(* IEC 61131-3 sources: SmartHomeNew/snapshots/2026-05-04, 69 files *)

(* ---- E_Behavior_Mode.dut ---- *)
TYPE E_Behavior_Mode :
(
    BEHAVIOR_HOME := 0,
    BEHAVIOR_AWAY := 1,
    BEHAVIOR_NIGHT := 2,
    BEHAVIOR_MAINTENANCE := 3
);
END_TYPE

(* ---- E_System_Reason_Code.dut ---- *)
{attribute 'strict'}
TYPE E_System_Reason_Code :
(
    REASON_NONE := 0,
    REASON_USER := 1,
    REASON_SAFETY := 2,
    REASON_AUTOMATION := 3,
    REASON_INTERNAL := 4,
    REASON_SCENARIO_VENT_BOOST := 5,
    REASON_USER_REQUEST := 6,
    REASON_SCENARIO_NIGHT := 7,
    REASON_DOMAIN_PROJECTION := 8
) USINT;
END_TYPE

(* ---- ST_Diagnostic_Event.dut ---- *)
{attribute 'pack_mode' := '1'}
TYPE ST_Diagnostic_Event :
STRUCT
    Code : UDINT;
    Severity : INT; // 1=info, 2=warning, 3=alarm, 4=critical
    Active : BOOL;
    Timestamp : UDINT;
    Source : INT; // producer/subsystem/index encoded by caller
END_STRUCT
END_TYPE

(* ---- ST_Operator_Zone_Rights.dut ---- *)
{attribute 'pack_mode' := '1'}
TYPE ST_Operator_Zone_Rights :
STRUCT
    operator_id : STRING(10);
    global_access_level : BYTE := 0;
    zone_masks : DWORD; // Битовая маска доступа к зонам (до 32 зон)
    last_modified : UDINT;
END_STRUCT
END_TYPE

(* ---- ST_System_Diagnostics.dut ---- *)
{attribute 'pack_mode' := '1'}
TYPE ST_System_Diagnostics :
STRUCT
    Freeze_Hardware_Event_Pending : BOOL;
    Freeze_Hardware_Event_Text : STRING(200);
    Backup_Pump_Fault : BOOL;
    Electric_Heater_Fault : BOOL;
    Backup_Pump_Recovered_After_Retry : BOOL;
    Electric_Heater_Recovered_After_Retry : BOOL;
    Backup_Pump_Out_Of_Service : BOOL;
    Electric_Heater_Out_Of_Service : BOOL;

    Pump_Exercise_Active : BOOL;
    Pump_Exercise_Failed : BOOL;
    Pump_Exercise_Last_Equipment : STRING(80);
    Pump_Exercise_Last_Result : STRING(120);
    Pump_Exercise_No_Feedback_Count : INT;
    Manifold_Pump_Exercise_Count : ARRAY[1..GVL_CONSTANTS.C_MAX_MANIFOLDS] OF UDINT;
    DHW_Heating_Pump_Exercise_Count : UDINT;
    DHW_Circ_Pump_Exercise_Count : UDINT;
    Backup_Pump_Exercise_Count : UDINT;
    Pump_Exercise_Event_Seq : UDINT;
    Pump_Exercise_Journal_1 : STRING(200);
    Pump_Exercise_Journal_2 : STRING(200);
    Pump_Exercise_Journal_3 : STRING(200);
    Pump_Exercise_Journal_Last_Seq : UDINT;

    Pump_Maintenance_Required : BOOL;
    Pump_Maintenance_Warning : BOOL;

    Manifold_Pump_Out_Of_Service : ARRAY[1..GVL_CONSTANTS.C_MAX_MANIFOLDS] OF BOOL;
    DHW_Heating_Pump_Out_Of_Service : BOOL;
    DHW_Circ_Pump_Out_Of_Service : BOOL;

    Maintenance_Last_Action : STRING(120);
    Operator_Action_Blocked : BOOL;
    Operator_Block_Reason : STRING(160);
    Operator_Last_Forbidden_Action : STRING(160);
    Operator_Journal_1 : STRING(200);
    Operator_Journal_2 : STRING(200);
    Operator_Journal_3 : STRING(200);
    Operator_Journal_Event_Seq : UDINT;
    Operator_Journal_Last_Seq : UDINT;

    Dangerous_Action_Pending_Confirm : BOOL;
    Dangerous_Action_Confirm_Text : STRING(160);
    Dangerous_Action_Confirm_Deadline_MS : UDINT;
    User_Access_Level_Active : INT;
    User_Access_Denied : BOOL;
    User_Access_Deny_Reason : STRING(160);

    Valve_Test_Mode_Active : BOOL;
    Valve_Test_Deadline_MS : UDINT;
    Valve_Test_Remaining_MS : UDINT;
    Valve_Test_Validation_OK : BOOL;
    Valve_Test_Validation_Text : STRING(160);
    Valve_Test_Forced_Close : BOOL;

    Water_Valve_Test_Mode_Active : BOOL;
    Water_Valve_Test_Deadline_MS : UDINT;
    Water_Valve_Test_Remaining_MS : UDINT;
    Water_Valve_Test_Validation_OK : BOOL;
    Water_Valve_Test_Validation_Text : STRING(160);
    Water_Valve_Test_Forced_Close : BOOL;
    Gas_Valve_Test_Mode_Active : BOOL;
    Gas_Valve_Test_Deadline_MS : UDINT;
    Gas_Valve_Test_Remaining_MS : UDINT;
    Gas_Valve_Test_Validation_OK : BOOL;
    Gas_Valve_Test_Validation_Text : STRING(160);
    Gas_Valve_Test_Forced_Close : BOOL;

    Active_Leak_Sensor_Index : INT;
    Active_Gas_Sensor_Index : INT;
    Active_Leak_Zone_Name : STRING(80);
    Active_Gas_Zone_Name : STRING(80);
    Water_Valve_Test_Context : STRING(160);
    Gas_Valve_Test_Context : STRING(160);

    Water_Recovery_Target_Zone_Index : INT;
    Gas_Recovery_Target_Zone_Index : INT;
    Water_Recovery_Selective_Allowed : BOOL;
    Gas_Recovery_Selective_Allowed : BOOL;
    Water_Recovery_Selective_Text : STRING(160);
    Gas_Recovery_Selective_Text : STRING(160);
    Water_Recovery_Physical_Active : BOOL;
    Water_Recovery_Physical_Zone_Name : STRING(80);

    Water_Zone_Open_Fault : ARRAY[1..32] OF BOOL;
    Water_Zone_Close_Fault : ARRAY[1..32] OF BOOL;
    Water_Valve_Exercise_Last_Zone : INT;
    Water_Valve_Exercise_Last_Result : STRING(160);
    Water_Zone_Critical_Close_Fault : ARRAY[1..32] OF BOOL;
    Water_Close_Fault_Active : BOOL;
    Water_Close_Fault_Zone_Name : STRING(80);
    Water_Close_Fault_Text : STRING(200);
    Water_Zone_Close_Retry_Active : ARRAY[1..32] OF BOOL;
    Water_Zone_Close_Retry_Count : ARRAY[1..32] OF INT;
    Water_Zone_Close_Recovered_After_Retry : ARRAY[1..32] OF BOOL;
    Water_Localization_Failed : BOOL;
    Water_Main_Shutdown_Recommended : BOOL;
    Water_Escalation_Text : STRING(200);
    Alarm_Event_Pulse : BOOL;
    Alarm_Event_Code : UDINT;
    Alarm_Event_Value : REAL;
    Sensor_Fault : BOOL;
    IO_Offline : BOOL;
    Subsystem_Degraded : BOOL;

    Manifold_Pressure_Fault : ARRAY[1..GVL_CONSTANTS.C_MAX_MANIFOLDS] OF BOOL;
    Manifold_Pressure_Diag_Code : ARRAY[1..GVL_CONSTANTS.C_MAX_MANIFOLDS] OF WORD;
    Manifold_Pressure_Fault_Active : BOOL;
    Manifold_Pressure_First_Fault_Index : INT;
    Manifold_Pressure_Fault_Text : STRING(160);

    Manifold_Current_Fault : ARRAY[1..GVL_CONSTANTS.C_MAX_MANIFOLDS] OF BOOL;
    Manifold_Current_Diag_Code : ARRAY[1..GVL_CONSTANTS.C_MAX_MANIFOLDS] OF WORD;
    Manifold_Current_Fault_Active : BOOL;
    Manifold_Current_First_Fault_Index : INT;
    Manifold_Current_Fault_Text : STRING(160);

    Manifold_Return_Temp_Fault : ARRAY[1..GVL_CONSTANTS.C_MAX_MANIFOLDS] OF BOOL;
    Manifold_Return_Temp_Diag_Code : ARRAY[1..GVL_CONSTANTS.C_MAX_MANIFOLDS] OF WORD;
    Manifold_Return_Temp_Fault_Active : BOOL;
    Manifold_Return_Temp_First_Fault_Index : INT;
    Manifold_Return_Temp_Fault_Text : STRING(160);

    Manifold_Sensor_Fault_Count : ARRAY[1..GVL_CONSTANTS.C_MAX_MANIFOLDS] OF INT;
    Manifold_Sensor_Out_Of_Service : ARRAY[1..GVL_CONSTANTS.C_MAX_MANIFOLDS] OF BOOL;
    Manifold_Sensor_Out_Of_Service_Active : BOOL;
    Manifold_Sensor_First_OOS_Index : INT;
    Manifold_Sensor_OOS_Text : STRING(160);
END_STRUCT
END_TYPE

(* ---- ST_Ventilation_Global_Config.dut ---- *)
{attribute 'pack_mode' := '1'}
TYPE ST_Ventilation_Global_Config :
STRUCT
    enable_ventilation : BOOL := TRUE;
    total_units : BYTE := 8;
    default_supply_speed : BYTE := 40;
    default_exhaust_speed : BYTE := 40;
    Degraded_Exhaust_Limit : BYTE := 30; // Ограничение вытяжки в режиме DEGRADED
    Scenario_Modes : ARRAY[1..GVL_CONSTANTS.C_MAX_SCENARIOS] OF ST_Ventilation_Scenario_Mode;
    wet_zone_to_exhaust_map : ARRAY[1..GVL_CONSTANTS.C_MAX_WET_ZONES] OF INT := [2, 3, 4, 5]; // Привязка мокрых зон к вытяжным вентиляторам
    pv3_exhaust_index : INT := 3; // Индекс вытяжного вентилятора ПВ-3
END_STRUCT
END_TYPE\n// VENT_POLICY_APPLIED
PolicyApplied : BOOL := TRUE;

(* ---- GVL_BEHAVIOR_ADAPT.gvl ---- *)
VAR_GLOBAL
    G_Behavior_Weights : ST_Behavior_Weights := (
        W_Comfort := 1.0,
        W_Night := 1.0,
        W_Preheat := 1.0,
        W_VentBoost := 1.0,
        W_AccessSecure := 1.0
    );

    G_Scenario_Stats : ARRAY[0..10] OF ST_Scenario_Stats;
    G_VentBoost_Zone_Adapt : ARRAY[1..GVL_CONSTANTS.C_MAX_ZONES] OF ST_Zone_Adapt_State;

    G_Adapt_Profile : E_Adapt_Profile := ADAPT_PROFILE_BALANCED;

    G_Adapt_Enabled : BOOL := TRUE;
    G_Adapt_Learning_Rate : REAL := 0.05;
    G_Adapt_Update_Threshold : INT := 5;

    G_Adapt_Min_Confidence : REAL := 0.30;
    G_Adapt_Default_Zone_Weight : REAL := 1.0;

    G_Confidence_Learning_Rate : REAL := 0.05;
    G_Decay_Factor : REAL := 0.995;

    G_Prev_Humidity : ARRAY[1..GVL_CONSTANTS.C_MAX_ZONES] OF REAL;
    G_Prev_Valid : ARRAY[1..GVL_CONSTANTS.C_MAX_ZONES] OF BOOL;
END_VAR
// >>> BULK_SYNC_ANCHOR: GVL_BEHAVIOR_ADAPT <<<

(* ---- GVL_COMMAND.gvl ---- *)
{attribute 'qualified_only'}
VAR_GLOBAL
    G_Gas_Valve_Close : BOOL := FALSE;
    G_Boiler_Stop : BOOL := FALSE;
    G_Supply_100_Req : BOOL := FALSE;
    G_Supply_80_Req : BOOL := FALSE;
    G_Vent_PV3_Boost : BOOL := FALSE;
    G_Exhaust_100_Req : BOOL := FALSE;
    G_Vent_Stop : BOOL := FALSE;
    G_Close_Valve_35 : BOOL := FALSE;
    G_Close_Valve_36 : BOOL := FALSE;
    G_Gate_Open : BOOL;
    G_Wicket_Open : BOOL;
    G_Lock_1_Open : BOOL;
    G_Lock_1_Close : BOOL;
    G_Lock_2_Open : BOOL;
    G_Lock_2_Close : BOOL;
    G_Reset_Errors : BOOL := FALSE;
    G_Scenario_Request : E_SCENARIO_TYPE := E_SCENARIO_TYPE.SCENARIO_NONE;
    G_Scenario_Request_Operator : E_SCENARIO_TYPE := E_SCENARIO_TYPE.SCENARIO_NONE;

    G_Arm_Req : BOOL;
    G_Disarm_Req : BOOL;
    G_PIN_Code : STRING(4);
    G_RFID_Tag : STRING(20);
    G_2FA_Code_In : STRING(6);
    G_Send_2FA_Req : BOOL;
    G_2FA_Code_Out : STRING(6);
    G_Lighting_Override : ARRAY[1..GVL_CONSTANTS.C_MAX_LIGHT_ZONES] OF BYTE;
    G_Blinds_Override : ARRAY[1..GVL_CONSTANTS.C_MAX_BLINDS] OF BYTE;
    G_Socket_Override : ARRAY[1..GVL_CONSTANTS.C_MAX_SOCKETS] OF BOOL;
    CMD_Set_Manifold_Pump_In_Service : ARRAY[1..GVL_CONSTANTS.C_MAX_MANIFOLDS] OF BOOL;
    CMD_Set_DHW_Heating_Pump_In_Service : BOOL;
    CMD_Set_DHW_Circ_Pump_In_Service : BOOL;
    CMD_Dangerous_Action_Confirm : BOOL;
    CMD_Dangerous_Action_Request : BOOL;
    CMD_User_Access_Level : INT := 0;
    CMD_Valve_Test_Open : BOOL;
    CMD_Valve_Test_Close : BOOL;
    CMD_Valve_Test_Confirm : BOOL;
    CMD_Water_Valve_Test_Open : BOOL;
    CMD_Water_Valve_Test_Close : BOOL;
    CMD_Water_Valve_Test_Confirm : BOOL;
    CMD_Gas_Valve_Test_Open : BOOL;
    CMD_Gas_Valve_Test_Close : BOOL;
    CMD_Gas_Valve_Test_Confirm : BOOL;
    CMD_Water_Selective_Recover : BOOL;
    CMD_Gas_Selective_Recover : BOOL;
END_VAR

(* ---- GVL_CONFIG.gvl ---- *)
{attribute 'qualified_only'}
VAR_GLOBAL
    // Subsystem Configurations
    G_Heating_Config : ST_Heating_Config; // Настройки системы отопления
    G_Ventilation_Config : ST_Ventilation_Config; // Настройки системы вентиляции
    G_DHW_Config : ST_DHW_Config; // Настройки горячего водоснабжения
    G_Security_Config : ST_Security_Global_Config; // Настройки системы безопасности
    G_Flood_Config : ST_Flood_Config; // Настройки системы защиты от протечек

    // HMI Configurations
    G_HMI_FloorHeating_Configs : ARRAY[1..GVL_CONSTANTS.C_MAX_HEATING_CIRCUITS] OF ST_FloorHeating_Circuit_Config; // Конфигурации контуров теплого пола
    G_Heating_Circuit_To_Zone : ARRAY[1..GVL_CONSTANTS.C_MAX_HEATING_CIRCUITS] OF INT := [1, 2, 3, 4, 5, 6, 7, 8, 9, 10, 11, 12, 13, 14, 15, 16]; // ВРЕМЕННО: circuit -> zone mapping, требует уточнения по фактической таблице помещений
    G_Wet_Zone_Map : ARRAY[1..32] OF BOOL; // Карта мокрых зон (TRUE = мокрая зона)
    G_HMI_Tariff_Settings : ST_Tariff_Config; // Настройки тарифов
    G_HMI_Vent_Global_Config : ST_Ventilation_Global_Config; // Глобальные настройки вентиляции
    G_HMI_Vent_Unit_Configs : ARRAY[1..GVL_CONSTANTS.C_MAX_VENT_UNITS] OF ST_Ventilation_Unit_Config; // Конфигурации отдельных вентустановок
    G_HMI_Scenario_Configs : ARRAY[1..GVL_CONSTANTS.C_MAX_SCENARIOS] OF ST_Scenario_Config; // Конфигурации сценариев
    G_HMI_Outdoor_Configs : ARRAY[1..GVL_CONSTANTS.C_MAX_OUTDOOR_ZONES] OF ST_Outdoor_Zone_Config; // Конфигурации зон уличного освещения
    G_HMI_Flood_Config : ST_Flood_Global_Config; // Глобальные настройки защиты от протечек
    G_HMI_Gas_Config : ST_Gas_Valve_Configuration; // Конфигурация системы газового контроля
    G_HMI_Sensor_Calibrations : ARRAY[1..GVL_CONSTANTS.C_MAX_CALIBRATIONS] OF ST_Sensor_Calibration_Record; // Данные калибровки датчиков
    G_HMI_User_Rules : ARRAY[1..GVL_CONSTANTS.C_MAX_RULES] OF ST_User_Rule; // Пользовательские правила (Rule Engine)

    // Sensor calibration pipeline
    G_Enable_Sensor_Calibration : BOOL := TRUE;
    G_Calib_Outdoor_Temp : ST_Sensor_Calibration_Record;
    G_Calib_Supply_Temps : ARRAY[1..GVL_CONSTANTS.C_MAX_SUPPLY_TEMPS] OF ST_Sensor_Calibration_Record;
    G_Calib_Room_Temps : ARRAY[1..GVL_CONSTANTS.C_MAX_ZONES] OF ST_Sensor_Calibration_Record;
    G_Calib_Floor_Temps : ARRAY[1..GVL_CONSTANTS.C_MAX_ZONES] OF ST_Sensor_Calibration_Record;
    G_Calib_CO2 : ARRAY[1..GVL_CONSTANTS.C_MAX_ZONES] OF ST_Sensor_Calibration_Record;
    G_Calib_Humidity : ARRAY[1..GVL_CONSTANTS.C_MAX_ZONES] OF ST_Sensor_Calibration_Record;
    G_Calib_Manifold_T_Supply : ARRAY[1..GVL_CONSTANTS.C_MAX_MANIFOLDS] OF ST_Sensor_Calibration_Record;
    G_Calib_Manifold_T_Return : ARRAY[1..GVL_CONSTANTS.C_MAX_MANIFOLDS] OF ST_Sensor_Calibration_Record;
    G_Calib_Methane : ARRAY[1..GVL_CONSTANTS.C_MAX_METHANE_SENSORS] OF ST_Sensor_Calibration_Record;
    G_Calib_CO : ARRAY[1..GVL_CONSTANTS.C_MAX_CO_SENSORS] OF ST_Sensor_Calibration_Record;

    // Конфигурация тестирования клапанов
    G_Valve_Test_Config : ARRAY[1..GVL_CONSTANTS.C_MAX_MANIFOLDS] OF ST_Valve_Test_Config;

    // HMI Commands & States
    G_HMI_Cleaning_Mode_Active : ARRAY[1..GVL_CONSTANTS.C_MAX_CLEANING_MODES] OF BOOL; // Режим уборки активен
    G_HMI_Cleaning_Mode_TimeLeft : ARRAY[1..GVL_CONSTANTS.C_MAX_CLEANING_MODES] OF UINT; // Оставшееся время режима уборки
    G_HMI_Admin_2FA_Enabled : BOOL := FALSE; // Включена ли 2FA для ADMIN
    G_HMI_Current_Operator_Factor2_Done : BOOL; // Второй фактор пройден
    G_HMI_Current_Operator_ID : STRING(10); // ID текущего оператора
    G_HMI_Manual_Gas_Valve_Open : BOOL; // Ручное открытие газового клапана
    G_HMI_Manual_Gas_Valve_Time : UDINT := 5; // Время ручного открытия
    G_HMI_Manual_Gas_Valve_TimeLeft : UDINT; // Оставшееся время ручного открытия
    G_HMI_Apply_Settings : BOOL; // Команда: Применить настройки
    G_HMI_Mute_Alarm : BOOL; // Команда: Временное отключение сирены
    G_HMI_Ack_Alarms : BOOL; // Команда: Квитировать все тревоги

    // Access Control Commands
    G_HMI_Gate_Open_Req : BOOL; // Запрос на открытие въездных ворот
    G_HMI_Wicket_Open_Req : BOOL; // Запрос на открытие калитки
    G_HMI_Lock_1_Open_Req : BOOL; // Разблокировка основного замка
    G_HMI_Lock_1_Close_Req : BOOL; // Блокировка основного замка
    G_HMI_Lock_2_Open_Req : BOOL; // Разблокировка доп. замка
    G_HMI_Lock_2_Close_Req : BOOL; // Блокировка доп. замка

    // HMI Settings
    G_HMI_Language : BYTE := 0; // 0=RU, 1=EN
    G_HMI_Brightness : BYTE := 80;
    G_HMI_Screen_Saver_Timeout : UDINT := 300; // сек

    // Сетевая безопасность
    G_Allowed_IPs : ARRAY[1..GVL_CONSTANTS.C_MAX_ALLOWED_IPS] OF STRING(15) := ['192.168.1.100','192.168.1.101','127.0.0.1','','']; // Разрешенные IP-адреса для шлюза

    G_Backup_Circulation_Pump_In_Service : BOOL := TRUE; // Резервный насос доступен для логики
    G_Electric_Heater_In_Service : BOOL := TRUE; // Электронагреватель доступен для логики
    G_Freeze_Hardware_Retry_Count : INT := 2; // Количество повторных попыток для anti-freeze hardware
    G_Freeze_Hardware_Retry_Delay_MS : UDINT := 5000; // Задержка между попытками повторного пуска
    G_Pump_Exercise_Enabled : BOOL := TRUE; // Разрешение периодической прокрутки насосов после простоя
    G_Pump_Exercise_Interval_MS : UDINT := 604800000; // 7 суток
    G_Pump_Exercise_Duration_MS : UDINT := 30000; // 30 сек
    G_Manifold_Pump_In_Service : ARRAY[1..GVL_CONSTANTS.C_MAX_MANIFOLDS] OF BOOL := [TRUE, TRUE, TRUE, TRUE, TRUE];
    G_Manifold_Priority : ARRAY[1..GVL_CONSTANTS.C_MAX_MANIFOLDS] OF INT := [3, 3, 2, 2, 1]; // 3=high, 2=normal, 1=low
    G_Manifold_Thermal_Weight : ARRAY[1..GVL_CONSTANTS.C_MAX_MANIFOLDS] OF REAL := [1.0, 1.0, 0.8, 0.8, 0.5];
    G_Max_Active_Manifolds : INT := 3; // energy-management limit for simultaneous active manifolds
    G_Max_Thermal_Budget : REAL := 6.0; // simplified manifold thermal budget units
    G_Policy_Min_Hold_MS : UDINT := 300000; // 5 min heating policy anti-oscillation hold
    G_DHW_Heating_Pump_In_Service : BOOL := TRUE;
    G_DHW_Circ_Pump_In_Service : BOOL := TRUE;
    G_Water_Valve_Exercise_Enabled : BOOL := TRUE;
    G_Water_Valve_Exercise_Interval_MS : UDINT := 604800000;
    G_Water_Valve_Exercise_Duration_MS : UDINT := 15000;
    G_Water_Valve_Exercise_Window_Start : TOD := TOD#04:00;
    G_Water_Valve_Exercise_Window_End : TOD := TOD#05:00;
    G_Water_Valve_Close_Retry_Count : INT := 2;
    G_Water_Valve_Close_Retry_Delay_MS : UDINT := 3000;
    // IO Mapping
    G_FloorTemp_Map : ARRAY[1..GVL_CONSTANTS.C_MAX_HEATING_CIRCUITS] OF INT := [1, 2, 3, 4, 5, 6, 7, 8, 9, 10, 11, 12, 13, 14, 15, 16];
    G_RoomTemp_Map : ARRAY[1..16] OF INT := [1, 2, 3, 4, 5, 6, 7, 8, 9, 10, 11, 12, 13, 14, 15, 16];
    G_Door_Map : ARRAY[1..GVL_CONSTANTS.C_MAX_DOOR_SENSORS] OF INT := [1, 2, 3, 4, 5, 6, 7, 8];
    G_Window_Map : ARRAY[1..16] OF INT := [9, 10, 11, 12, 13, 14, 15, 16, 17, 18, 19, 20, 21, 22, 23, 24];

    // Evacuation config
    C_MAX_LIGHT_ZONES : INT := 32; // fallback if not defined elsewhere
    G_Evac_Exit_Zones : ARRAY[1..32] OF BOOL; // зоны-выходы (TRUE = выход)
    G_Evac_Smoke_Zone_Map : ARRAY[1..GVL_CONSTANTS.C_MAX_SMOKE_SENSORS] OF INT; // Привязка дымовых датчиков к зонам эвакуации
    G_Evac_Leak_Zone_Map : ARRAY[1..GVL_CONSTANTS.C_MAX_FLOOD_SENSORS] OF INT; // Привязка датчиков протечки к зонам эвакуации
    G_Evac_Gas_Zone_Map : ARRAY[1..GVL_CONSTANTS.C_MAX_METHANE_SENSORS] OF INT; // Привязка газовых датчиков к зонам эвакуации
    G_Evac_Zone_Names : ARRAY[1..32] OF STRING(80); // Человекочитаемые имена зон (помещения/крыло/этаж/сторона)

END_VAR

VAR_GLOBAL CONSTANT
    C_MS_PER_SEC    : UDINT := GVL_CONSTANTS.C_MS_IN_SECOND; // Миллисекунд в секунду
    C_SEC_PER_MIN   : UDINT := 60; // Секунд в минуту
    C_MIN_PER_HOUR  : UDINT := 60; // Минут в часе
    C_MS_PER_MIN    : UDINT := GVL_CONSTANTS.C_MS_IN_MINUTE; // Миллисекунд в минуту
    C_MAX_RULES     : INT := 20; // Максимальное количество пользовательских правил
    C_ZONE_COUNT    : BYTE := 18; // Общее количество зон в системе

    // Коды ошибок
    ERR_PRESSURE_OUT_OF_RANGE : UDINT := 16#E004;
    ERR_HIGH_DELTA_T : UDINT := 16#E005;
    ERR_BOILER_OFFLINE : UDINT := 16#E006;
    ERR_BOILER_GENERAL_FAULT : UDINT := 16#E007;
    ERR_BOILER_NO_FLAME : UDINT := 16#E008;
    ERR_PUMP_NO_CURRENT : UDINT := 16#E009;
    ERR_PUMP_UNDERCURRENT : UDINT := 16#E00A;
    ERR_PUMP_OVERCURRENT : UDINT := 16#E00B;
    ERR_DELTA_T_LOW : UDINT := 16#E00C;
    ERR_DELTA_T_HIGH : UDINT := 16#E00D;
    ERR_DHW_IO_OFFLINE : UDINT := 16#E00E;
    ERR_DHW_TEMP_SENSOR_FAULT : UDINT := 16#E00F;
    ERR_DHW_PRESSURE_OUT_OF_RANGE : UDINT := 16#E010;
    ERR_DHW_PRESSURE_SENSOR_FAULT : UDINT := 16#E011;
    ERR_BACKUP_PUMP_OUT_OF_SERVICE : UDINT := 16#E012;
    ERR_ELECTRIC_HEATER_OUT_OF_SERVICE : UDINT := 16#E013;
    ERR_MANIFOLD_PUMP_OUT_OF_SERVICE : UDINT := 16#E014;
    ERR_DHW_HEATING_PUMP_OUT_OF_SERVICE : UDINT := 16#E015;
    ERR_DHW_CIRC_PUMP_OUT_OF_SERVICE : UDINT := 16#E016;
    ERR_FREEZE_HARDWARE_FAILED : UDINT := 16#E017;
END_VAR

(* ---- GVL_CONFIG_SIMULATION.gvl ---- *)
{attribute 'qualified_only'}
VAR_GLOBAL
    G_Simulation_Request : BOOL := FALSE;
    G_Simulation_Confirm : BOOL := FALSE;
    G_Simulation_Result_OK : BOOL := TRUE;
    G_Simulation_Error_Text : STRING(200) := '';
    G_Simulation_Last_Run_MS : UDINT := 0;
END_VAR

(* ---- GVL_CONFIG_VALIDATION.gvl ---- *)
{attribute 'qualified_only'}
VAR_GLOBAL
    G_Config_Valid : BOOL := TRUE;
    G_Config_Auto_Corrected : BOOL := FALSE;
    G_Config_Reset_To_Default_Done : BOOL := FALSE;
    G_Config_Last_Error_Text : STRING(200) := '';
    G_Config_Last_Action_Text : STRING(200) := '';
    G_Config_Last_Update_MS : UDINT := 0;
END_VAR

(* ---- GVL_DIAGNOSTICS_EXT.gvl ---- *)
{attribute 'qualified_only'}
VAR_GLOBAL
    // Health scores (0..1)
    G_Health_Heating : REAL := 1.0;
    G_Health_Safety : REAL := 1.0;
    G_Health_IO : REAL := 1.0;

    // Error counters
    G_Error_Count_Heating : UDINT := 0;
    G_Error_Count_Safety : UDINT := 0;
    G_Error_Count_IO : UDINT := 0;

    // Last error timestamps
    G_Last_Error_Time_Heating : UDINT := 0;
    G_Last_Error_Time_Safety : UDINT := 0;
    G_Last_Error_Time_IO : UDINT := 0;

    // Timing
    G_Last_Update_Time : UDINT := 0;

    // States
    G_Heating_State : INT := 0; // 0=OK,1=DEGRADED,2=CRITICAL
    G_Safety_State : INT := 0;
    G_IO_State : INT := 0;
END_VAR

(* ---- GVL_EVENT.gvl ---- *)
VAR_GLOBAL
    G_Event_Log : ARRAY[0..63] OF ST_EVENT;
    G_Event_Head : UINT;
    G_Event_ID_Counter : UDINT;
END_VAR

(* ---- GVL_INTENT_SAFETY.gvl ---- *)
VAR_GLOBAL
    // --- meta / traceability ---
    I_Source_Valid : BOOL := FALSE;
    I_Last_Update_Cycle : UDINT := 0;
    I_Last_Update_MS : UDINT := 0;

    // --- safety facts for arbitration ---
    I_Fire_Alarm_Active : BOOL := FALSE;
    I_Gas_Alarm_Active : BOOL := FALSE;
    I_Leak_Alarm_Active : BOOL := FALSE;
    I_CO_Warning_Active : BOOL := FALSE;
    I_System_Safe_Stop_Required : BOOL := FALSE;
    I_Freeze_Protection_Required : BOOL := FALSE;
    I_Evacuation_Mode_Active : BOOL := FALSE;

    // --- gas / boiler / ventilation constraints ---
    I_Gas_Close_Required : BOOL := FALSE;
    I_Boiler_Stop_Required : BOOL := FALSE;
    I_Vent_Stop_Required : BOOL := FALSE;
    I_Vent_Force_PV3_Boost : BOOL := FALSE;
    I_Vent_Force_Supply_100 : BOOL := FALSE;
    I_Vent_Force_Supply_80 : BOOL := FALSE;
    I_Vent_Force_Exhaust_100 : BOOL := FALSE;

    // --- water constraints ---
    I_Water_Main_Close_Required : BOOL := FALSE;
    I_Water_Zone_Close_Required : ARRAY[1..32] OF BOOL;
    I_Water_Selective_Recovery_Allowed : BOOL := FALSE;
    I_Water_Recovery_Target_Zone : INT := 0;

    // --- lock / evacuation constraints ---
    I_Lock_1_Force_Open : BOOL := FALSE;
    I_Lock_1_Force_Close_Block : BOOL := FALSE;
    I_Lock_2_Force_Open : BOOL := FALSE;
    I_Lock_2_Force_Close_Block : BOOL := FALSE;
END_VAR

(* ---- GVL_PRESENCE.gvl ---- *)
{attribute 'qualified_only'}
VAR_GLOBAL
    G_Any_Motion : BOOL := FALSE;
    G_Occupied : BOOL := TRUE;
    G_Auto_Away_Request : BOOL := FALSE;
    G_Last_Motion_TS : UDINT := 0;

    G_Zone_Occupied : ARRAY[1..GVL_CONSTANTS.C_MAX_ZONES] OF BOOL;
    G_Zone_Last_Motion_TS : ARRAY[1..GVL_CONSTANTS.C_MAX_ZONES] OF UDINT;
END_VAR

(* ---- GVL_Retain.gvl ---- *)
{attribute 'qualified_only'}
VAR_GLOBAL RETAIN
    G_Initialized : BOOL := FALSE; // Флаг инициализации retain-переменных

    // Энергонезависимая память (NVRAM) для хранения настроек и логов
    G_NVRAM_Data : ARRAY[0..12799] OF BYTE; // 100 * 128 = 12800 байт

    // Буфер черного ящика (100 записей)
    G_BlackBox_Buffer : ARRAY[0..GVL_CONSTANTS.C_MAX_BLACKBOX_RECORDS-1] OF ST_BlackBox_Record;
    G_BlackBox_LastIndex : INT;
    G_BlackBox_Frozen : BOOL;
    G_Presence_History : ARRAY[0..GVL_CONSTANTS.C_MAX_PRESENCE_HISTORY-1] OF WORD; // 168 часов * 6 записей в час = 1008 записей (битовая маска 16 ламп)

    // История событий
    G_History_Buffer : ARRAY[1..GVL_CONSTANTS.C_MAX_HISTORY_RECORDS] OF ST_History_Record;
    G_History_Write_Idx : INT := 1;
    G_History_Total_Events : UDINT;

    // Статистика котлов
    G_Boiler_Accumulated_MS : ARRAY[1..GVL_CONSTANTS.C_MAX_BOILERS] OF UDINT;
    G_Boiler_Work_Seconds : ARRAY[1..GVL_CONSTANTS.C_MAX_BOILERS] OF UDINT;

    // Результаты тестирования клапанов
    G_Valve_Test_Results : ARRAY[1..GVL_CONSTANTS.C_MAX_MANIFOLDS] OF BOOL;

    // ПИН-коды доступа (храним хэши CRC32 для безопасности)
    // 16#9BE3E0A3 - это CRC32 от строки '1234'
    G_Access_Codes : ARRAY[1..GVL_CONSTANTS.C_MAX_ACCESS_CODES] OF DWORD := [16#9BE3E0A3, 16#4A89A12D, 16#F4DBDF21, 16#90F59C65, 16#0972D346, 0, 0, 0, 0, 0];

    // Зарегистрированные RFID/NFC метки (строковое представление UID)
    G_RFID_Tags : ARRAY[1..GVL_CONSTANTS.C_MAX_ACCESS_CODES] OF STRING(20) := ['A1B2C3D4', 'E5F67890', '', '', '', '', '', '', '', ''];
END_VAR

(* ---- IValveController.st ---- *)
INTERFACE IValveController
METHOD OpenValve : BOOL
VAR_INPUT
    VI_Operator_ID : STRING(10);
    VI_Force : BOOL;
END_VAR
END_METHOD

METHOD CloseValve : BOOL
VAR_INPUT
    VI_Operator_ID : STRING(10);
    VI_Force : BOOL;
END_VAR
END_METHOD

METHOD GetStatus : BYTE
END_METHOD
END_INTERFACE

(* ---- FB_Analog_Validator.st ---- *)
FUNCTION_BLOCK FB_Analog_Validator
VAR_INPUT
    VI_Value : REAL;
    VI_Min_Valid : REAL;
    VI_Max_Valid : REAL;
    VI_Fallback_Mode : INT := 0; // 0: Hold last good, 1: Default value
    VI_Default_Value : REAL := 0.0;
END_VAR
VAR_OUTPUT
    VO_Value : REAL;
    VO_Error : BOOL;
END_VAR
VAR
    L_Last_Good_Value : REAL;
    L_First_Valid : BOOL := FALSE;
END_VAR

IF VI_Value >= VI_Min_Valid AND VI_Value <= VI_Max_Valid THEN
    VO_Error := FALSE;
    VO_Value := VI_Value;
    L_Last_Good_Value := VI_Value;
    L_First_Valid := TRUE;
ELSE
    VO_Error := TRUE;
    IF VI_Fallback_Mode = 1 OR NOT L_First_Valid THEN
        VO_Value := VI_Default_Value;
    ELSE
        VO_Value := L_Last_Good_Value;
    END_IF;
END_IF;
// >>> BULK_SYNC_ANCHOR: FB_Analog_Validator <<<

(* ---- FB_Device_Predictive_Diag.st ---- *)
FUNCTION_BLOCK FB_Device_Predictive_Diag
VAR_INPUT
    VI_Current_Value : REAL;      // Текущий ток или время
    VI_Nominal_Value : REAL;      // Эталонное значение
    VI_Is_Running    : BOOL;
    VI_Reset_Stats   : BOOL;
    VI_System_Time_MS: UDINT;     // Системное время (мс)
END_VAR
VAR_IN_OUT
    VIO_Health_Data  : ST_Device_Health;
END_VAR
VAR
    L_Prev_Running   : BOOL;
    L_Start_Time     : UDINT;
    L_Last_Calc_Time : UDINT;
    L_Elapsed_MS     : UDINT;
    L_Accumulated_MS : UDINT; // Накопленное время работы (мс)
    L_Timer_Running  : FB_System_Timer;
END_VAR

// 0. Сброс статистики
IF VI_Reset_Stats THEN
    VIO_Health_Data.Starts_Count := 0;
    VIO_Health_Data.Sample_Count := 0;
    VIO_Health_Data.Current_Sum := 0.0;
    VIO_Health_Data.Avg_Start_Current := 0.0;
    VIO_Health_Data.Health_Score := 100;
    VIO_Health_Data.Maintenance_Required := FALSE;
    VIO_Health_Data.Warning_Message := '';
    VIO_Health_Data.Last_Start_Current := 0.0;
    VIO_Health_Data.Total_Runtime_Hours := 0;
    L_Accumulated_MS := 0;
END_IF;

// 1. Счётчик пусков и замер пускового тока
IF VI_Is_Running AND NOT L_Prev_Running THEN
    VIO_Health_Data.Starts_Count := VIO_Health_Data.Starts_Count + 1;
    VIO_Health_Data.Last_Start_Current := VI_Current_Value;
    L_Start_Time := VI_System_Time_MS;
    L_Last_Calc_Time := VI_System_Time_MS;

    // Обновление среднего пускового тока
    VIO_Health_Data.Sample_Count := VIO_Health_Data.Sample_Count + 1;
    VIO_Health_Data.Current_Sum := VIO_Health_Data.Current_Sum + VI_Current_Value;
    VIO_Health_Data.Avg_Start_Current := VIO_Health_Data.Current_Sum / UDINT_TO_REAL(VIO_Health_Data.Sample_Count);

    // 2. Анализ отклонения пускового тока (п. 12.1 ТЗ)
    IF VI_Current_Value > (VI_Nominal_Value * 1.5) THEN
        VIO_Health_Data.Health_Score := TO_BYTE(LIMIT(0, TO_INT(VIO_Health_Data.Health_Score) - 5, 100));
    ELSIF VI_Current_Value > (VI_Nominal_Value * 1.2) THEN
        VIO_Health_Data.Health_Score := TO_BYTE(LIMIT(0, TO_INT(VIO_Health_Data.Health_Score) - 1, 100));
    ELSIF VI_Current_Value < (VI_Nominal_Value * 0.5) THEN
        VIO_Health_Data.Health_Score := TO_BYTE(LIMIT(0, TO_INT(VIO_Health_Data.Health_Score) - 2, 100));
    END_IF;
END_IF;

// 3. Анализ рабочего тока и наработки
IF VI_Is_Running THEN
    L_Elapsed_MS := (VI_System_Time_MS - L_Last_Calc_Time);
    L_Accumulated_MS := L_Accumulated_MS + L_Elapsed_MS;
    L_Last_Calc_Time := VI_System_Time_MS;

    // Обновляем наработку каждый час (3600000 мс)
    IF L_Accumulated_MS >= 3600000 THEN
        VIO_Health_Data.Total_Runtime_Hours := VIO_Health_Data.Total_Runtime_Hours + 1;
        L_Accumulated_MS := L_Accumulated_MS - 3600000;

        // Естественный износ: -1% здоровья каждые 1000 часов
        IF (VIO_Health_Data.Total_Runtime_Hours MOD 1000) = 0 THEN
            VIO_Health_Data.Health_Score := TO_BYTE(LIMIT(0, TO_INT(VIO_Health_Data.Health_Score) - 1, 100));
        END_IF;

        // Анализ рабочего тока (после пускового режима)
        IF (VI_System_Time_MS - L_Start_Time) > 10000 THEN // 10 секунд после пуска
            IF VI_Current_Value > (VI_Nominal_Value * 1.1) THEN
                // Повышенный рабочий ток - ускоренный износ (-1% в час)
                VIO_Health_Data.Health_Score := TO_BYTE(LIMIT(0, TO_INT(VIO_Health_Data.Health_Score) - 1, 100));
            END_IF;
        END_IF;
    END_IF;
END_IF;

// 4. Генерация предупреждения
IF VIO_Health_Data.Health_Score < 20 THEN
    VIO_Health_Data.Maintenance_Required := TRUE;
    VIO_Health_Data.Warning_Message := 'Критический износ: проверьте механику';
ELSIF VIO_Health_Data.Health_Score < 60 THEN
    VIO_Health_Data.Maintenance_Required := FALSE;
    VIO_Health_Data.Warning_Message := 'Предупреждение: повышенное трение';
ELSE
    VIO_Health_Data.Maintenance_Required := FALSE;
    VIO_Health_Data.Warning_Message := 'В норме';
END_IF;

L_Prev_Running := VI_Is_Running;

(* ---- FB_Diagnostics_Event_Manager.st ---- *)
FUNCTION_BLOCK FB_Diagnostics_Event_Manager
VAR_INPUT
    VI_Code : UDINT;
    VI_Severity : INT;
    VI_Active : BOOL;
    VI_Timestamp : UDINT;
    VI_Source : INT;
END_VAR
VAR_IN_OUT
    VIO_Events : ARRAY[1..50] OF ST_Diagnostic_Event;
    VIO_Count : INT;
END_VAR
VAR
    L_Index : INT;
    L_i : INT;
    L_Found_Index : INT;
    L_Was_Active : BOOL;
    L_Debounce_Index : INT;
    L_Oldest_Index : INT;
    L_Oldest_Time : UDINT;
    L_Stable_State : BOOL;

    L_Debounce_Used : ARRAY[1..50] OF BOOL;
    L_Debounce_Code : ARRAY[1..50] OF UDINT;
    L_Debounce_Source : ARRAY[1..50] OF INT;
    L_Debounce_Last_Input_State : ARRAY[1..50] OF BOOL;
    L_Debounce_Stable_State : ARRAY[1..50] OF BOOL;
    L_Debounce_Last_Change_Time : ARRAY[1..50] OF UDINT;
END_VAR

L_Found_Index := 0;
L_Was_Active := FALSE;
FOR L_i := 1 TO 50 DO
    IF (VIO_Events[L_i].Code = VI_Code) AND (VIO_Events[L_i].Source = VI_Source) THEN
        L_Found_Index := L_i;
        L_Was_Active := VIO_Events[L_i].Active;
        EXIT;
    END_IF;
END_FOR;

L_Debounce_Index := 0;
L_Oldest_Time := 16#FFFFFFFF;
L_Oldest_Index := 1;

FOR L_i := 1 TO 50 DO
    IF L_Debounce_Used[L_i] THEN
        IF (L_Debounce_Code[L_i] = VI_Code) AND (L_Debounce_Source[L_i] = VI_Source) THEN
            L_Debounce_Index := L_i;
            EXIT;
        END_IF;
        IF L_Debounce_Last_Change_Time[L_i] < L_Oldest_Time THEN
            L_Oldest_Time := L_Debounce_Last_Change_Time[L_i];
            L_Oldest_Index := L_i;
        END_IF;
    ELSE
        L_Debounce_Index := L_i;
        EXIT;
    END_IF;
END_FOR;

IF L_Debounce_Index = 0 THEN
    L_Debounce_Index := L_Oldest_Index;
END_IF;

IF NOT L_Debounce_Used[L_Debounce_Index] OR
   (L_Debounce_Code[L_Debounce_Index] <> VI_Code) OR
   (L_Debounce_Source[L_Debounce_Index] <> VI_Source) THEN
    L_Debounce_Used[L_Debounce_Index] := TRUE;
    L_Debounce_Code[L_Debounce_Index] := VI_Code;
    L_Debounce_Source[L_Debounce_Index] := VI_Source;
    L_Debounce_Last_Input_State[L_Debounce_Index] := VI_Active;
    L_Debounce_Stable_State[L_Debounce_Index] := FALSE;
    L_Debounce_Last_Change_Time[L_Debounce_Index] := VI_Timestamp;
END_IF;

IF VI_Active <> L_Debounce_Last_Input_State[L_Debounce_Index] THEN
    L_Debounce_Last_Input_State[L_Debounce_Index] := VI_Active;
    L_Debounce_Last_Change_Time[L_Debounce_Index] := VI_Timestamp;
END_IF;

IF (VI_Timestamp - L_Debounce_Last_Change_Time[L_Debounce_Index]) > 2000 THEN
    L_Debounce_Stable_State[L_Debounce_Index] := L_Debounce_Last_Input_State[L_Debounce_Index];
END_IF;

L_Stable_State := L_Debounce_Stable_State[L_Debounce_Index];

IF L_Stable_State THEN
    IF NOT L_Was_Active THEN
        L_Index := (VIO_Count MOD 50) + 1;
        VIO_Events[L_Index].Code := VI_Code;
        VIO_Events[L_Index].Severity := VI_Severity;
        VIO_Events[L_Index].Active := TRUE;
        VIO_Events[L_Index].Timestamp := VI_Timestamp;
        VIO_Events[L_Index].Source := VI_Source;
        VIO_Count := VIO_Count + 1;
    ELSIF L_Found_Index > 0 THEN
        VIO_Events[L_Found_Index].Severity := VI_Severity;
    END_IF;
ELSE
    IF L_Found_Index > 0 THEN
        VIO_Events[L_Found_Index].Active := FALSE;
    END_IF;
END_IF;

// >>> BULK_SYNC_ANCHOR: FB_Diagnostics_Event_Manager <<<

(* ---- FB_Diagnostics_RootCause.st ---- *)
FUNCTION_BLOCK FB_Diagnostics_RootCause
VAR_INPUT
    VI_Emergency_Stop : BOOL;
    VI_Gas_Safety : BOOL;
    VI_IO_Failsafe : BOOL;

    VI_Boiler_OT_Online : ARRAY[1..GVL_CONSTANTS.C_MAX_BOILERS] OF BOOL;
    VI_Boiler_Error : ARRAY[1..GVL_CONSTANTS.C_MAX_BOILERS] OF BOOL;
    VI_Boiler_Flame : ARRAY[1..GVL_CONSTANTS.C_MAX_BOILERS] OF BOOL;

    VI_Manifold_Pumps : ARRAY[1..GVL_CONSTANTS.C_MAX_MANIFOLDS] OF BOOL;
    VI_Manifold_Valves : ARRAY[1..GVL_CONSTANTS.C_MAX_MANIFOLDS] OF REAL;

    VI_Sensor_Error : BOOL;

    VI_Supply_Temps : ARRAY[1..GVL_CONSTANTS.C_MAX_MANIFOLDS] OF REAL;
    VI_Target_Supply : REAL;

    VI_Demand_Map : ARRAY[1..GVL_CONSTANTS.C_MAX_MANIFOLDS] OF BOOL;
END_VAR

VAR_OUTPUT
    VO_RootCause : E_Heating_RootCause;
    VO_Confidence : REAL;
END_VAR

VAR
    L_i : INT;
    L_AnyBoilerOnline : BOOL;
    L_AnyBoilerError : BOOL;
    L_AnyFlame : BOOL;
    L_AnyDemand : BOOL;
    L_AnyPumpOn : BOOL;
    L_AnyValveOpen : BOOL;
    L_LowSupply : BOOL;
END_VAR

// --- Safety ---
IF VI_Emergency_Stop THEN
    VO_RootCause := E_Heating_RootCause.RC_EMERGENCY_STOP;
    VO_Confidence := 1.0;
    RETURN;
END_IF;

IF VI_Gas_Safety THEN
    VO_RootCause := E_Heating_RootCause.RC_GAS_SAFETY;
    VO_Confidence := 1.0;
    RETURN;
END_IF;

IF VI_IO_Failsafe THEN
    VO_RootCause := E_Heating_RootCause.RC_IO_OFFLINE;
    VO_Confidence := 1.0;
    RETURN;
END_IF;

// --- Aggregate flags ---
L_AnyBoilerOnline := FALSE;
L_AnyBoilerError := FALSE;
L_AnyFlame := FALSE;

FOR L_i := 1 TO GVL_CONSTANTS.C_MAX_BOILERS DO
    IF VI_Boiler_OT_Online[L_i] THEN L_AnyBoilerOnline := TRUE; END_IF;
    IF VI_Boiler_Error[L_i] THEN L_AnyBoilerError := TRUE; END_IF;
    IF VI_Boiler_Flame[L_i] THEN L_AnyFlame := TRUE; END_IF;
END_FOR;

L_AnyDemand := FALSE;
L_AnyPumpOn := FALSE;
L_AnyValveOpen := FALSE;
L_LowSupply := FALSE;

FOR L_i := 1 TO GVL_CONSTANTS.C_MAX_MANIFOLDS DO
    IF VI_Demand_Map[L_i] THEN L_AnyDemand := TRUE; END_IF;
    IF VI_Manifold_Pumps[L_i] THEN L_AnyPumpOn := TRUE; END_IF;
    IF VI_Manifold_Valves[L_i] > 5.0 THEN L_AnyValveOpen := TRUE; END_IF;
    IF VI_Supply_Temps[L_i] < (VI_Target_Supply - 2.0) THEN L_LowSupply := TRUE; END_IF;
END_FOR;

// --- Boiler ---
IF NOT L_AnyBoilerOnline THEN
    VO_RootCause := E_Heating_RootCause.RC_BOILER_OFFLINE;
    VO_Confidence := 0.9;
    RETURN;
END_IF;

IF L_AnyBoilerError THEN
    VO_RootCause := E_Heating_RootCause.RC_BOILER_ERROR;
    VO_Confidence := 0.9;
    RETURN;
END_IF;

IF NOT L_AnyFlame THEN
    VO_RootCause := E_Heating_RootCause.RC_NO_FLAME;
    VO_Confidence := 0.8;
    RETURN;
END_IF;

// --- Hydraulics ---
IF L_AnyDemand THEN
    IF NOT L_AnyPumpOn THEN
        VO_RootCause := E_Heating_RootCause.RC_PUMP_FAILURE;
        VO_Confidence := 0.8;
        RETURN;
    END_IF;

    IF NOT L_AnyValveOpen THEN
        VO_RootCause := E_Heating_RootCause.RC_VALVES_CLOSED;
        VO_Confidence := 0.8;
        RETURN;
    END_IF;
END_IF;

// --- Thermal ---
IF L_AnyDemand AND L_LowSupply THEN
    VO_RootCause := E_Heating_RootCause.RC_NO_HEAT_TRANSFER;
    VO_Confidence := 0.7;
    RETURN;
END_IF;

// --- Sensors ---
IF VI_Sensor_Error THEN
    VO_RootCause := E_Heating_RootCause.RC_SENSOR_ERROR;
    VO_Confidence := 0.7;
    RETURN;
END_IF;

VO_RootCause := E_Heating_RootCause.RC_NONE;
VO_Confidence := 0.0;

END_FUNCTION_BLOCK

(* ---- FB_FloorHeating_Freeze_Protection.st ---- *)
FUNCTION_BLOCK FB_FloorHeating_Freeze_Protection
VAR_INPUT
    VI_Outdoor_Temp : REAL;
    VI_Threshold : REAL := 7.0;
END_VAR
VAR_IN_OUT
    VI_Floor_Temps : ARRAY[1..GVL_CONSTANTS.C_MAX_HEATING_CIRCUITS] OF REAL;
END_VAR
VAR_OUTPUT
    VO_Freeze_Alert : BOOL;
    VO_Pump_Force_On : BOOL;
END_VAR
VAR
    L_i : INT;
END_VAR

VO_Freeze_Alert := FALSE;
VO_Pump_Force_On := FALSE;

FOR L_i := 1 TO GVL_CONSTANTS.C_MAX_HEATING_CIRCUITS DO
    IF VI_Floor_Temps[L_i] < VI_Threshold THEN
        VO_Freeze_Alert := TRUE;
        VO_Pump_Force_On := TRUE;
        RETURN;
    END_IF;
END_FOR;

IF VI_Outdoor_Temp < -5.0 THEN
    VO_Pump_Force_On := TRUE;
END_IF;
END_FUNCTION_BLOCK

(* ---- FB_Heating_Execution_Core.st ---- *)
FUNCTION_BLOCK FB_Heating_Execution_Core
VAR_INPUT
    VI_System_Time_MS : UDINT;
    VI_Current_TOD : TOD;
    VI_Current_Day_Of_Week : UINT;
    VI_IsActivePLC : BOOL;
    VI_Outdoor_Temp : REAL;
    VI_Floor_Temps : ARRAY[1..GVL_CONSTANTS.C_MAX_HEATING_CIRCUITS] OF REAL;
    VI_Room_Temps : ARRAY[1..GVL_CONSTANTS.C_MAX_ZONES] OF REAL;
    VI_Config : ST_Heating_Config;
    VI_Zone_Configs : ARRAY[1..GVL_CONSTANTS.C_MAX_HEATING_CIRCUITS] OF ST_FloorHeating_Circuit_Config;
    VI_Tariff : ST_Tariff_Config;
    VI_Time_Of_Day_MS : UDINT;
    VI_Manifold_Pressures : ARRAY[1..GVL_CONSTANTS.C_MAX_MANIFOLDS] OF REAL;
    VI_Manifold_Currents : ARRAY[1..GVL_CONSTANTS.C_MAX_MANIFOLDS] OF REAL;
    VI_Manifold_Temps_Supply : ARRAY[1..GVL_CONSTANTS.C_MAX_MANIFOLDS] OF REAL;
    VI_Manifold_Temps_Return : ARRAY[1..GVL_CONSTANTS.C_MAX_MANIFOLDS] OF REAL;
    VI_Boiler_Flame_Status : ARRAY[1..GVL_CONSTANTS.C_MAX_BOILERS] OF BOOL;
    VI_Boiler_Error_Status : ARRAY[1..GVL_CONSTANTS.C_MAX_BOILERS] OF BOOL;
    VI_Boiler_OT_Online : ARRAY[1..GVL_CONSTANTS.C_MAX_BOILERS] OF BOOL;
    VI_Boiler_Modulation : ARRAY[1..GVL_CONSTANTS.C_MAX_BOILERS] OF REAL;
    VI_Rule_Actions : ARRAY[1..GVL_CONSTANTS.C_MAX_RULES] OF ST_Rule_Action;
    VI_IO_Modules_Online : ARRAY[1..GVL_CONSTANTS.C_MAX_MODULES] OF BOOL;
    VI_DHW_Heating_Demand : BOOL;
    VI_DHW_Target_Temp : REAL;
    VI_DHW_Temp : REAL;
    VI_DHW_Pressure : REAL;
    VI_DHW_Config : ST_DHW_Config;
    VI_Reset_Errors : BOOL;
    VI_System_Mode : E_System_Operating_Mode;
    VI_Emergency_Stop : BOOL;
    VI_Gas_Safety_Stop : BOOL;
    VI_Manifold_End_Switches : ARRAY[1..GVL_CONSTANTS.C_MAX_MANIFOLDS] OF BOOL;
    VI_Valve_Test_Config : ARRAY[1..GVL_CONSTANTS.C_MAX_MANIFOLDS] OF ST_Valve_Test_Config;
END_VAR
VAR_IN_OUT
    VIO_Manifold_Valves : ARRAY[1..GVL_CONSTANTS.C_MAX_MANIFOLDS] OF REAL;
    VIO_Manifold_Pumps : ARRAY[1..GVL_CONSTANTS.C_MAX_MANIFOLDS] OF BOOL;
    VIO_Zone_Valves : ARRAY[1..GVL_CONSTANTS.C_MAX_HEATING_CIRCUITS] OF BOOL;
    VIO_Boiler_OT_Enable : ARRAY[1..GVL_CONSTANTS.C_MAX_BOILERS] OF BOOL;
    VIO_Boiler_OT_Setpoint : ARRAY[1..GVL_CONSTANTS.C_MAX_BOILERS] OF REAL;
    VIO_Backup_Circulation_Pump : BOOL;
    VIO_Electric_Heater_Enable : BOOL;
    VIO_Freeze_Risk_Status : BOOL;
    VIO_Manifold_Status : ARRAY[1..GVL_CONSTANTS.C_MAX_MANIFOLDS] OF ST_Manifold_Status;
    VIO_Boiler_Status : ARRAY[1..GVL_CONSTANTS.C_MAX_BOILERS] OF ST_Boiler_Status;
    VIO_DHW_Heating_Pump : BOOL;
    VIO_DHW_Circ_Pump : BOOL;
    VIO_DHW_Status : ST_DHW_Status;
END_VAR
VAR
    fbHeatingManager : FB_Heating_System_Manager;
    fbDHWManager : FB_DHW_Manager;
END_VAR

// Pure execution core: calls heating and DHW managers.
// Does not apply command/allocation overrides.

fbHeatingManager(
    VI_System_Time_MS := VI_System_Time_MS,
    VI_IsActivePLC := VI_IsActivePLC,
    VI_Outdoor_Temp := VI_Outdoor_Temp,
    VI_Floor_Temps := VI_Floor_Temps,
    VI_Room_Temps := VI_Room_Temps,
    VI_Config := VI_Config,
    VI_Zone_Configs := VI_Zone_Configs,
    VI_Tariff := VI_Tariff,
    VI_Current_Hour := TO_UINT(VI_Time_Of_Day_MS / GVL_CONSTANTS.C_MS_IN_HOUR),
    VI_Manifold_Pressures := VI_Manifold_Pressures,
    VI_Manifold_Currents := VI_Manifold_Currents,
    VI_Manifold_Temps_Supply := VI_Manifold_Temps_Supply,
    VI_Manifold_Temps_Return := VI_Manifold_Temps_Return,
    VI_Boiler_Flame_Status := VI_Boiler_Flame_Status,
    VI_Boiler_Error_Status := VI_Boiler_Error_Status,
    VI_Boiler_OT_Online := VI_Boiler_OT_Online,
    VI_Boiler_Modulation := VI_Boiler_Modulation,
    VI_Rule_Actions := VI_Rule_Actions,
    VI_IO_Modules_Online := VI_IO_Modules_Online,
    VI_DHW_Heating_Demand := VI_DHW_Heating_Demand,
    VI_DHW_Target_Temp := VI_DHW_Target_Temp,
    VI_System_Mode := VI_System_Mode,
    VI_Emergency_Stop := VI_Emergency_Stop,
    VI_Gas_Safety_Stop := VI_Gas_Safety_Stop,
    VI_Manifold_End_Switches := VI_Manifold_End_Switches,
    VI_Valve_Test_Config := VI_Valve_Test_Config,
    VO_Manifold_Valves => VIO_Manifold_Valves,
    VO_Manifold_Pumps => VIO_Manifold_Pumps,
    VO_Zone_Valves => VIO_Zone_Valves,
    VO_Boiler_OT_Enable => VIO_Boiler_OT_Enable,
    VO_Boiler_OT_Setpoint => VIO_Boiler_OT_Setpoint,
    VO_Backup_Circulation_Pump => VIO_Backup_Circulation_Pump,
    VO_Electric_Heater_Enable => VIO_Electric_Heater_Enable,
    VO_Freeze_Risk_Status => VIO_Freeze_Risk_Status,
    VO_Status => VIO_Manifold_Status,
    VO_Boiler_Status => VIO_Boiler_Status
);

fbDHWManager(
    VI_System_Time_MS := VI_System_Time_MS,
    VI_Current_TOD := VI_Current_TOD,
    VI_IsActivePLC := VI_IsActivePLC,
    VI_Temp := VI_DHW_Temp,
    VI_Pressure := VI_DHW_Pressure,
    VI_Config := VI_DHW_Config,
    VI_Current_Day_Of_Week := VI_Current_Day_Of_Week,
    VI_IO_Modules_Online := VI_IO_Modules_Online,
    VI_Reset_Errors := VI_Reset_Errors,
    VI_Emergency_Stop := VI_Emergency_Stop,
    VI_System_Mode := VI_System_Mode,
    VO_Heating_Pump => VIO_DHW_Heating_Pump,
    VO_Circ_Pump => VIO_DHW_Circ_Pump,
    VO_Status => VIO_DHW_Status
);

END_FUNCTION_BLOCK
// >>> BULK_SYNC_ANCHOR: FB_Heating_Execution_Core <<<

(* ---- FB_Heating_Optimizer.st ---- *)
FUNCTION_BLOCK FB_Heating_Optimizer
VAR
    L_i : INT;
    L_Load : REAL;
    L_Total_Demand : REAL;
END_VAR

L_Total_Demand := 0.0;

// calculate total demand
FOR L_i := 1 TO GVL_CONSTANTS.C_MAX_ZONES DO
    L_Total_Demand := L_Total_Demand + ABS(GVL_HEATING_POLICY.G_Zone_Thermal_Demand[L_i]);
END_FOR;

GVL_HEATING_POLICY.G_Optimization_Load_Index := L_Total_Demand;

// normalize and optimize
FOR L_i := 1 TO GVL_CONSTANTS.C_MAX_ZONES DO

    IF L_Total_Demand > 0.01 THEN
        L_Load := ABS(GVL_HEATING_POLICY.G_Zone_Thermal_Demand[L_i]) / L_Total_Demand;
    ELSE
        L_Load := 0.0;
    END_IF;

    // priority score
    GVL_HEATING_POLICY.G_Zone_Optimization_Score[L_i] :=
        L_Load +
        (1.0 - GVL_HEATING_POLICY.G_Zone_Thermal_Model_Confidence[L_i]) * 0.2;

    // load balancing: reduce low priority zones
    IF GVL_HEATING_POLICY.G_Zone_Optimization_Score[L_i] < 0.2 THEN
        GVL_HEATING_POLICY.G_Zone_Thermal_Demand[L_i] :=
            GVL_HEATING_POLICY.G_Zone_Thermal_Demand[L_i] * 0.5;
    END_IF;

    // peak shaving
    IF L_Total_Demand > 5.0 THEN
        GVL_HEATING_POLICY.G_Zone_Thermal_Demand[L_i] :=
            GVL_HEATING_POLICY.G_Zone_Thermal_Demand[L_i] * 0.7;
        GVL_HEATING_POLICY.G_Optimization_Energy_Saving_Active := TRUE;
    END_IF;

END_FOR;

END_FUNCTION_BLOCK

(* ---- FB_Heating_Safe_State.st ---- *)
FUNCTION_BLOCK FB_Heating_Safe_State
VAR_INPUT
    VI_Block_Normal_Heating : BOOL;
    VI_IO_Failsafe_Active : BOOL;
    VI_Gas_Safety_Active : BOOL;
    VI_Freeze_Active : BOOL;
    VI_Freeze_Target_Supply : REAL;
    VI_Manifold_Temps_Supply : ARRAY[1..GVL_CONSTANTS.C_MAX_MANIFOLDS] OF REAL;
    VI_Boiler_Error_Status : ARRAY[1..GVL_CONSTANTS.C_MAX_BOILERS] OF BOOL;
    VI_Boiler_OT_Online : ARRAY[1..GVL_CONSTANTS.C_MAX_BOILERS] OF BOOL;
END_VAR
VAR_OUTPUT
    VO_Applied : BOOL;
    VO_Zone_Valves : ARRAY[1..GVL_CONSTANTS.C_MAX_HEATING_CIRCUITS] OF BOOL;
    VO_Manifold_Pumps : ARRAY[1..GVL_CONSTANTS.C_MAX_MANIFOLDS] OF BOOL;
    VO_Manifold_Valves : ARRAY[1..GVL_CONSTANTS.C_MAX_MANIFOLDS] OF REAL;
    VO_Boiler_OT_Enable : ARRAY[1..GVL_CONSTANTS.C_MAX_BOILERS] OF BOOL;
    VO_Boiler_OT_Setpoint : ARRAY[1..GVL_CONSTANTS.C_MAX_BOILERS] OF REAL;
    VO_Boiler_Status : ARRAY[1..GVL_CONSTANTS.C_MAX_BOILERS] OF ST_Boiler_Status;
    VO_Backup_Circulation_Pump : BOOL;
    VO_Electric_Heater_Enable : BOOL;
    VO_Freeze_Risk_Status : BOOL;
END_VAR
VAR
    L_i : INT;
    L_Min_Supply_Temp : REAL;
END_VAR

VO_Applied := VI_Block_Normal_Heating;
VO_Backup_Circulation_Pump := FALSE;
VO_Electric_Heater_Enable := FALSE;
VO_Freeze_Risk_Status := FALSE;

IF NOT VI_Block_Normal_Heating THEN
    RETURN;
END_IF;

FOR L_i := 1 TO GVL_CONSTANTS.C_MAX_HEATING_CIRCUITS DO
    VO_Zone_Valves[L_i] := FALSE;
END_FOR;

FOR L_i := 1 TO GVL_CONSTANTS.C_MAX_MANIFOLDS DO
    IF VI_IO_Failsafe_Active AND VI_Freeze_Active THEN
        VO_Manifold_Pumps[L_i] := TRUE;
        VO_Manifold_Valves[L_i] := 35.0;
    ELSE
        VO_Manifold_Pumps[L_i] := FALSE;
        VO_Manifold_Valves[L_i] := 0.0;
    END_IF;
END_FOR;

FOR L_i := 1 TO GVL_CONSTANTS.C_MAX_BOILERS DO
    VO_Boiler_OT_Enable[L_i] := FALSE;
    VO_Boiler_OT_Setpoint[L_i] := 0.0;
    VO_Boiler_Status[L_i].Warning := FALSE;
    VO_Boiler_Status[L_i].Error := TRUE;
END_FOR;

IF VI_Gas_Safety_Active AND VI_Freeze_Active THEN
    VO_Backup_Circulation_Pump := TRUE;
    L_Min_Supply_Temp := 1000.0;
    FOR L_i := 1 TO GVL_CONSTANTS.C_MAX_MANIFOLDS DO
        IF VI_Manifold_Temps_Supply[L_i] < L_Min_Supply_Temp THEN
            L_Min_Supply_Temp := VI_Manifold_Temps_Supply[L_i];
        END_IF;
    END_FOR;
    IF L_Min_Supply_Temp > 900.0 THEN
        L_Min_Supply_Temp := 0.0;
    END_IF;

    IF L_Min_Supply_Temp < (VI_Freeze_Target_Supply - 1.0) THEN
        VO_Electric_Heater_Enable := TRUE;
    ELSIF L_Min_Supply_Temp > (VI_Freeze_Target_Supply + 1.0) THEN
        VO_Electric_Heater_Enable := FALSE;
    END_IF;
    VO_Freeze_Risk_Status := TRUE;
END_IF;

IF VI_IO_Failsafe_Active AND VI_Freeze_Active THEN
    IF VI_Boiler_OT_Online[1] AND NOT VI_Boiler_Error_Status[1] THEN
        VO_Boiler_OT_Enable[1] := TRUE;
        VO_Boiler_OT_Setpoint[1] := VI_Freeze_Target_Supply;
    END_IF;
END_IF;

END_FUNCTION_BLOCK
// >>> BULK_SYNC_ANCHOR: FB_Heating_Safe_State <<<

(* ---- FB_Heating_Safety_Gate.st ---- *)
// ==============================================================================
// Heating safety gate helper
// ==============================================================================
FUNCTION_BLOCK FB_Heating_Safety_Gate
VAR_INPUT
    VI_System_Mode : E_System_Operating_Mode;
    VI_Emergency_Stop : BOOL;
    VI_Gas_Safety_Stop : BOOL;
    VI_IO_Failsafe_Active : BOOL;
    VI_Outdoor_Temp : REAL;
    VI_Freeze_Threshold : REAL;
END_VAR

VAR_IN_OUT
    VI_Floor_Temps : ARRAY[1..GVL_CONSTANTS.C_MAX_HEATING_CIRCUITS] OF REAL;
END_VAR

VAR_OUTPUT
    VO_Block_Normal_Heating : BOOL;
    VO_Gas_Safety_Active : BOOL;
    VO_Emergency_Safe_Stop_Active : BOOL;
    VO_IO_Failsafe_Active : BOOL;
    VO_Freeze_Mode_Active : BOOL;
    VO_Freeze_Target_Supply : REAL;
    VO_Outdoor_Temp_Valid : BOOL;
END_VAR

VAR
    L_i : INT;
    L_Outdoor_Temp_Safe : REAL;
END_VAR

VO_Gas_Safety_Active := VI_Gas_Safety_Stop;
VO_Emergency_Safe_Stop_Active := VI_Emergency_Stop OR (VI_System_Mode = E_System_Operating_Mode.MODE_SAFE_STOP);
VO_IO_Failsafe_Active := VI_IO_Failsafe_Active;

// REAL validity guard: NaN fails self-equality; extreme values are rejected as sensor faults.
VO_Outdoor_Temp_Valid := (VI_Outdoor_Temp = VI_Outdoor_Temp) AND (VI_Outdoor_Temp > -80.0) AND (VI_Outdoor_Temp < 80.0);
IF VO_Outdoor_Temp_Valid THEN
    L_Outdoor_Temp_Safe := VI_Outdoor_Temp;
ELSE
    L_Outdoor_Temp_Safe := 20.0;
    GVL_STATE.G_Heating_Sensor_Fault := TRUE;
END_IF;

VO_Block_Normal_Heating := VO_Gas_Safety_Active OR VO_Emergency_Safe_Stop_Active OR VO_IO_Failsafe_Active;
VO_Freeze_Mode_Active := (VI_System_Mode = E_System_Operating_Mode.MODE_FREEZE_PROTECTION) OR (L_Outdoor_Temp_Safe < -5.0);

FOR L_i := 1 TO GVL_CONSTANTS.C_MAX_HEATING_CIRCUITS DO
    IF VI_Floor_Temps[L_i] < 7.0 THEN
        VO_Freeze_Mode_Active := TRUE;
    END_IF;
END_FOR;

IF VO_Freeze_Mode_Active THEN
    VO_Freeze_Target_Supply := LIMIT(20.0, VI_Freeze_Threshold + 2.0, 35.0);
ELSE
    VO_Freeze_Target_Supply := 0.0;
END_IF;

// >>> BULK_SYNC_ANCHOR: FB_Heating_Safety_Gate <<<

(* ---- FB_HMI_Interface.st ---- *)
FUNCTION_BLOCK FB_HMI_Interface
VAR_INPUT
    VI_Severity   : E_System_Severity;
    VI_RootCause  : E_System_Root_Cause;
    VI_Status_Msg : STRING(200);
END_VAR

VAR_OUTPUT
    VO_HMI_Status_Text : STRING(200);
    VO_HMI_State_Code  : INT;
END_VAR

VO_HMI_Status_Text := VI_Status_Msg;

CASE VI_Severity OF
    E_System_Severity.SEV_NORMAL:
        VO_HMI_State_Code := 0;
    E_System_Severity.SEV_WARNING:
        VO_HMI_State_Code := 1;
    E_System_Severity.SEV_DEGRADED:
        VO_HMI_State_Code := 2;
    E_System_Severity.SEV_CRITICAL:
        VO_HMI_State_Code := 3;
END_CASE;
// >>> BULK_SYNC_ANCHOR: FB_HMI_Interface <<<

(* ---- FB_Lifetime_Manager.st ---- *)
FUNCTION_BLOCK FB_Lifetime_Manager
VAR_INPUT
    VI_System_Time_MS : UDINT;
    VI_Device_Active  : BOOL;
    VI_Device_ID      : BYTE;
    VI_Nominal_Hours : UDINT;
END_VAR

VAR_IN_OUT
    VIO_Status : ST_Lifetime_Status;
END_VAR

VAR
    L_Last_Time : UDINT;
    L_Prev_State : BOOL;
    L_Delta_MS : UDINT;
    L_Runtime_Accum_MS : UDINT;
    L_Remaining_Percent_UDINT : UDINT;
END_VAR

// === DELTA TIME ===
IF VI_System_Time_MS >= L_Last_Time THEN
    L_Delta_MS := VI_System_Time_MS - L_Last_Time;
ELSE
    // overflow
    L_Delta_MS := (4294967295 - L_Last_Time) + VI_System_Time_MS + 1;
END_IF;

L_Last_Time := VI_System_Time_MS;

// === START COUNT ===
IF VI_Device_Active AND NOT L_Prev_State THEN
    VIO_Status.start_count := VIO_Status.start_count + 1;
END_IF;

L_Prev_State := VI_Device_Active;

// === RUNTIME ACCUMULATION ===
IF VI_Device_Active THEN
    L_Runtime_Accum_MS := L_Runtime_Accum_MS + L_Delta_MS;

    WHILE L_Runtime_Accum_MS >= 3600000 DO
        VIO_Status.runtime_hours := VIO_Status.runtime_hours + 1;
        L_Runtime_Accum_MS := L_Runtime_Accum_MS - 3600000;
    END_WHILE;
END_IF;

// === BASIC LIFETIME ESTIMATION ===
IF VI_Nominal_Hours > 0 THEN
    IF VIO_Status.runtime_hours >= VI_Nominal_Hours THEN
        VIO_Status.remaining_hours := 0;
        VIO_Status.remaining_percent := 0;
    ELSE
        VIO_Status.remaining_hours := VI_Nominal_Hours - VIO_Status.runtime_hours;
        L_Remaining_Percent_UDINT := (VIO_Status.remaining_hours * 100) / VI_Nominal_Hours;

        IF L_Remaining_Percent_UDINT > 100 THEN
            L_Remaining_Percent_UDINT := 100;
        END_IF;

        VIO_Status.remaining_percent := UDINT_TO_BYTE(L_Remaining_Percent_UDINT);
    END_IF;
ELSE
    VIO_Status.remaining_hours := 0;
    VIO_Status.remaining_percent := 0;
END_IF;

VIO_Status.maintenance_required := VIO_Status.remaining_percent <= GVL_Lifetime.G_Maintenance_Threshold_Percent;

// === BASIC FLAGS ===
VIO_Status.device_id := VI_Device_ID;
VIO_Status.last_calc_timestamp := VI_System_Time_MS;

END_FUNCTION_BLOCK

(* ---- FB_Maintenance_Access.st ---- *)
FUNCTION_BLOCK FB_Maintenance_Access
VAR_INPUT
    VI_System_Time : UDINT;
    VI_Activate    : BOOL;
    VI_Duration    : UDINT := 60; // мин
END_VAR
VAR_OUTPUT
    VO_Active      : BOOL;
    VO_Time_Left   : UDINT;
END_VAR
VAR
    L_Start_Time   : UDINT;
    L_elapsed      : UDINT;
END_VAR

IF VI_Activate AND NOT VO_Active THEN
    VO_Active := TRUE;
    L_Start_Time := VI_System_Time;
END_IF;

IF VO_Active THEN
    L_elapsed := (SEL(VI_System_Time >= L_Start_Time, VI_System_Time - L_Start_Time, (4294967295 - L_Start_Time) + VI_System_Time + 1)) / GVL_CONSTANTS.C_MS_IN_MINUTE;
    IF L_elapsed >= VI_Duration THEN
        VO_Active := FALSE;
        VO_Time_Left := 0;
    ELSE
        VO_Time_Left := VI_Duration - L_elapsed;
    END_IF;
ELSE
    VO_Time_Left := 0;
END_IF;

(* ---- FB_Mode_Manager.st ---- *)
FUNCTION_BLOCK FB_Mode_Manager

VAR_INPUT
    VI_Is_Night : BOOL;
    VI_Away_Request : BOOL;
    VI_Maintenance_Request : BOOL;
    VI_System_Time_MS : UDINT;
END_VAR

VAR_OUTPUT
    VO_Mode : E_Behavior_Mode;
    VO_Mode_Code : UDINT;
END_VAR

// default
VO_Mode := BEHAVIOR_HOME;
VO_Mode_Code := 0;

// priority-based transitions
IF VI_Maintenance_Request THEN
    VO_Mode := BEHAVIOR_MAINTENANCE;
    VO_Mode_Code := 300;
ELSIF VI_Away_Request THEN
    VO_Mode := BEHAVIOR_AWAY;
    VO_Mode_Code := 200;
ELSIF VI_Is_Night THEN
    VO_Mode := BEHAVIOR_NIGHT;
    VO_Mode_Code := 100;
END_IF;

(* ---- FB_Persist_Pipeline.st ---- *)
FUNCTION_BLOCK FB_Persist_Pipeline
VAR_INPUT
    VI_PersistStruct : ST_Persist;
    VI_System_Time_MS : UDINT;
    VI_IsActivePLC : BOOL;
END_VAR
VAR_IN_OUT
    VIO_Apply_Settings : BOOL;
    VIO_Persist_Buffer : ARRAY[0..4] OF BYTE;
    VIO_Last_Written_Persist_Buffer : ARRAY[0..4] OF BYTE;
    VIO_Last_Persist_Write_MS : UDINT;
END_VAR
VAR_OUTPUT
    VO_NVRAM_Cmd : BYTE;
    VO_NVRAM_Offset : UDINT;
    VO_NVRAM_Done : BOOL;
    VO_NVRAM_Err : BOOL;
    VO_NVRAM_ErrID : UDINT;
END_VAR
VAR
    fbNVRAMManager : FB_NVRAM_Manager;
    L_Persist_Buffer_Changed : BOOL;
END_VAR

// === SERIALIZE PERSIST STRUCT → BUFFER ===

// System Mode
VIO_Persist_Buffer[0] := TO_BYTE(TO_INT(VI_PersistStruct.System_Mode));

// Gas
IF VI_PersistStruct.Safety_Gas_Latched THEN
    VIO_Persist_Buffer[1] := BYTE#1;
ELSE
    VIO_Persist_Buffer[1] := BYTE#0;
END_IF;

// Smoke
IF VI_PersistStruct.Safety_Smoke_Latched THEN
    VIO_Persist_Buffer[2] := BYTE#1;
ELSE
    VIO_Persist_Buffer[2] := BYTE#0;
END_IF;

// Leak
IF VI_PersistStruct.Safety_Leak_Latched THEN
    VIO_Persist_Buffer[3] := BYTE#1;
ELSE
    VIO_Persist_Buffer[3] := BYTE#0;
END_IF;

// DHW Pump
IF VI_PersistStruct.DHW_Heating_Pump THEN
    VIO_Persist_Buffer[4] := BYTE#1;
ELSE
    VIO_Persist_Buffer[4] := BYTE#0;
END_IF;

// === END SERIALIZE ===

L_Persist_Buffer_Changed :=
    (VIO_Persist_Buffer[0] <> VIO_Last_Written_Persist_Buffer[0]) OR
    (VIO_Persist_Buffer[1] <> VIO_Last_Written_Persist_Buffer[1]) OR
    (VIO_Persist_Buffer[2] <> VIO_Last_Written_Persist_Buffer[2]) OR
    (VIO_Persist_Buffer[3] <> VIO_Last_Written_Persist_Buffer[3]) OR
    (VIO_Persist_Buffer[4] <> VIO_Last_Written_Persist_Buffer[4]);

VO_NVRAM_Cmd := 0;
VO_NVRAM_Offset := 0;

IF VIO_Apply_Settings THEN
    // explicit config apply requests a controlled write
    // keep flag set until successful write confirmation
    VO_NVRAM_Cmd := 1;

ELSIF L_Persist_Buffer_Changed THEN
    // controlled write: no more often than once per 60 seconds
    IF (VIO_Last_Persist_Write_MS = 0) OR
       ((VI_System_Time_MS - VIO_Last_Persist_Write_MS) >= 60000) THEN
        VO_NVRAM_Cmd := 1;
    END_IF;
END_IF;

fbNVRAMManager(
    VI_Command := VO_NVRAM_Cmd,
    VI_Offset := VO_NVRAM_Offset,
    VI_DataRef := VIO_Persist_Buffer[0],
    VI_DataSize := 5,
    VI_System_Time_MS := VI_System_Time_MS,
    VI_Operator_ID := 'SYSTEM',
    VI_IsActivePLC := VI_IsActivePLC,
    VI_TwoPersonConfirmation := FALSE,
    VO_Done => VO_NVRAM_Done,
    VO_Error => VO_NVRAM_Err,
    VO_ErrorID => VO_NVRAM_ErrID
);

IF (VO_NVRAM_Cmd = 1) AND VO_NVRAM_Done AND NOT VO_NVRAM_Err THEN
    VIO_Last_Written_Persist_Buffer[0] := VIO_Persist_Buffer[0];
    VIO_Last_Written_Persist_Buffer[1] := VIO_Persist_Buffer[1];
    VIO_Last_Written_Persist_Buffer[2] := VIO_Persist_Buffer[2];
    VIO_Last_Written_Persist_Buffer[3] := VIO_Persist_Buffer[3];
    VIO_Last_Written_Persist_Buffer[4] := VIO_Persist_Buffer[4];
    VIO_Last_Persist_Write_MS := VI_System_Time_MS;
    VIO_Apply_Settings := FALSE;
END_IF;
END_FUNCTION_BLOCK

(* ---- FB_PID_Controller.st ---- *)
FUNCTION_BLOCK FB_PID_Controller
VAR_INPUT
    VI_SetPoint : REAL;
    VI_ProcessValue : REAL;
    VI_Kp : REAL;
    VI_Tn : REAL;
    VI_Tv : REAL;
    VI_Y_Min : REAL := REAL#0.0;
    VI_Y_Max : REAL := REAL#100.0;
    VI_Manual_Mode : BOOL;
    VI_Manual_Value : REAL;
    VI_Deadband : REAL := REAL#0.1;
    VI_Cycle_Time_S : REAL := REAL#0.01;
    VI_Reset : BOOL;
END_VAR
VAR_OUTPUT
    VO_Output : REAL;
    VO_Error : REAL;
    VO_Limiting : BOOL;
END_VAR
VAR
    L_Integral_Sum : REAL;
    L_Prev_Error : REAL;
    L_Derivative : REAL;
    L_P_Term : REAL;
    L_I_Candidate : REAL;
    L_D_Term : REAL;
    L_Output_Predicted : REAL;
    L_Output_Raw : REAL;
    L_Cycle_Time_Safe : REAL;
END_VAR

L_Cycle_Time_Safe := VI_Cycle_Time_S;
IF L_Cycle_Time_Safe <= REAL#0.0 THEN
    L_Cycle_Time_Safe := REAL#0.01;
END_IF;

VO_Error := VI_SetPoint - VI_ProcessValue;
IF ABS(VO_Error) < VI_Deadband THEN
    VO_Error := REAL#0.0;
END_IF;

IF VI_Reset THEN
    L_Integral_Sum := REAL#0.0;
    L_Prev_Error := REAL#0.0;
    VO_Output := LIMIT(VI_Y_Min, REAL#0.0, VI_Y_Max);
    VO_Limiting := FALSE;
    RETURN;
END_IF;

L_P_Term := VI_Kp * VO_Error;

IF VI_Tv > REAL#0.0 THEN
    L_Derivative := (VO_Error - L_Prev_Error) / L_Cycle_Time_Safe;
    L_D_Term := VI_Kp * VI_Tv * L_Derivative;
ELSE
    L_Derivative := REAL#0.0;
    L_D_Term := REAL#0.0;
END_IF;

IF VI_Manual_Mode THEN
    VO_Output := LIMIT(VI_Y_Min, VI_Manual_Value, VI_Y_Max);
    L_Integral_Sum := VO_Output - L_P_Term - L_D_Term;
    L_Prev_Error := VO_Error;
    VO_Limiting := (VO_Output <= VI_Y_Min) OR (VO_Output >= VI_Y_Max);
    RETURN;
END_IF;

IF VI_Tn > REAL#0.0 THEN
    L_I_Candidate := L_Integral_Sum + ((VI_Kp / VI_Tn) * VO_Error * L_Cycle_Time_Safe);
ELSE
    L_I_Candidate := L_Integral_Sum;
END_IF;

L_Output_Predicted := L_P_Term + L_I_Candidate + L_D_Term;

// Anti-windup: accept the new integral only if it does not push the output farther into saturation.
IF VI_Tn > REAL#0.0 THEN
    IF (L_Output_Predicted > VI_Y_Max) AND (VO_Error > REAL#0.0) THEN
        // hold integral
    ELSIF (L_Output_Predicted < VI_Y_Min) AND (VO_Error < REAL#0.0) THEN
        // hold integral
    ELSE
        L_Integral_Sum := L_I_Candidate;
    END_IF;
END_IF;

L_Output_Raw := L_P_Term + L_Integral_Sum + L_D_Term;
VO_Output := LIMIT(VI_Y_Min, L_Output_Raw, VI_Y_Max);
VO_Limiting := (L_Output_Raw > VI_Y_Max) OR (L_Output_Raw < VI_Y_Min);
L_Prev_Error := VO_Error;

// >>> BULK_SYNC_ANCHOR: FB_PID_Controller <<<
END_FUNCTION_BLOCK

(* ---- FB_Rule_Engine.st ---- *)
FUNCTION_BLOCK FB_Rule_Engine
VAR_INPUT
    VI_System_Time_MS : UDINT;
    VI_IsActivePLC : BOOL;
    VI_Security_Armed : BOOL;
    VI_Current_Time : TOD;
    VI_Day_Of_Week : INT;
END_VAR
VAR_IN_OUT
    VI_Rules : ARRAY[1..GVL_CONSTANTS.C_MAX_RULES] OF ST_User_Rule;
    VI_Indoor_Temps : ARRAY[1..16] OF REAL;
    VI_Floor_Temps : ARRAY[1..GVL_CONSTANTS.C_MAX_HEATING_CIRCUITS] OF REAL;
    VI_Humidities : ARRAY[1..16] OF REAL;
    VI_CO2_Levels : ARRAY[1..16] OF REAL;
    VI_Motion_Sensors : ARRAY[1..16] OF BOOL;
    VI_Door_Sensors : ARRAY[1..GVL_CONSTANTS.C_MAX_DOOR_SENSORS] OF BOOL;
    VI_Window_Sensors : ARRAY[1..16] OF BOOL;
    VI_Water_Sensors : ARRAY[1..GVL_CONSTANTS.C_MAX_FLOOD_SENSORS] OF BOOL;
    VI_Smoke_Sensors : ARRAY[1..GVL_CONSTANTS.C_MAX_SMOKE_SENSORS] OF BOOL;
    VI_Methane_Sensors : ARRAY[1..GVL_CONSTANTS.C_MAX_METHANE_SENSORS] OF REAL;
    VI_CO_Sensors : ARRAY[1..GVL_CONSTANTS.C_MAX_CO_SENSORS] OF REAL;
END_VAR
VAR_OUTPUT
    VO_Preheat_Request : BOOL;
    VO_Actions : ARRAY[1..GVL_CONSTANTS.C_MAX_RULES] OF ST_Rule_Action;
END_VAR
VAR
    L_i : INT;
    L_Condition_Met : BOOL;
    L_Current_Value : REAL;
    L_Triggers : ARRAY[1..GVL_CONSTANTS.C_MAX_RULES] OF R_TRIG;
    L_Trigger_Count : ARRAY[1..GVL_CONSTANTS.C_MAX_RULES] OF UINT;
    L_Last_Reset_Time : UDINT;
    L_Elapsed_Time : UDINT;
END_VAR

IF NOT VI_IsActivePLC THEN RETURN; END_IF;

VO_Preheat_Request := FALSE;

L_Elapsed_Time := SEL(VI_System_Time_MS >= L_Last_Reset_Time, VI_System_Time_MS - L_Last_Reset_Time, (4294967295 - L_Last_Reset_Time) + VI_System_Time_MS + 1);

IF L_Elapsed_Time >= GVL_CONSTANTS.C_MS_IN_MINUTE THEN
    L_Last_Reset_Time := VI_System_Time_MS;
    FOR L_i := 1 TO GVL_CONSTANTS.C_MAX_RULES DO
        L_Trigger_Count[L_i] := 0;
    END_FOR;
END_IF;

FOR L_i := 1 TO GVL_CONSTANTS.C_MAX_RULES DO

    VO_Actions[L_i].Active := FALSE;
    IF VI_Rules[L_i].Enabled THEN
        L_Condition_Met := FALSE;
        L_Current_Value := 0.0;

        IF VI_Rules[L_i].Condition_Target_ID > 0 THEN
            CASE VI_Rules[L_i].Condition_Type OF
                E_Rule_Condition_Type.COND_AIR_TEMP: IF VI_Rules[L_i].Condition_Target_ID <= 16 THEN L_Current_Value := VI_Indoor_Temps[VI_Rules[L_i].Condition_Target_ID]; END_IF;
                E_Rule_Condition_Type.COND_FLOOR_TEMP: IF VI_Rules[L_i].Condition_Target_ID <= GVL_CONSTANTS.C_MAX_HEATING_CIRCUITS THEN L_Current_Value := VI_Floor_Temps[VI_Rules[L_i].Condition_Target_ID]; END_IF;
                E_Rule_Condition_Type.COND_HUMIDITY: IF VI_Rules[L_i].Condition_Target_ID <= 16 THEN L_Current_Value := VI_Humidities[VI_Rules[L_i].Condition_Target_ID]; END_IF;
                E_Rule_Condition_Type.COND_CO2: IF VI_Rules[L_i].Condition_Target_ID <= 16 THEN L_Current_Value := VI_CO2_Levels[VI_Rules[L_i].Condition_Target_ID]; END_IF;
                E_Rule_Condition_Type.COND_MOTION: IF VI_Rules[L_i].Condition_Target_ID <= 16 THEN L_Current_Value := SEL(VI_Motion_Sensors[VI_Rules[L_i].Condition_Target_ID], 0.0, 1.0); END_IF;
                E_Rule_Condition_Type.COND_DOOR_WINDOW:
                    IF VI_Rules[L_i].Condition_Target_ID <= GVL_CONSTANTS.C_MAX_DOOR_SENSORS THEN
                        L_Current_Value := SEL(VI_Door_Sensors[VI_Rules[L_i].Condition_Target_ID] OR VI_Window_Sensors[VI_Rules[L_i].Condition_Target_ID], 0.0, 1.0);
                    ELSIF VI_Rules[L_i].Condition_Target_ID <= 16 THEN
                        L_Current_Value := SEL(VI_Window_Sensors[VI_Rules[L_i].Condition_Target_ID], 0.0, 1.0);
                    END_IF;
                E_Rule_Condition_Type.COND_FLOOD: IF VI_Rules[L_i].Condition_Target_ID <= GVL_CONSTANTS.C_MAX_FLOOD_SENSORS THEN L_Current_Value := SEL(VI_Water_Sensors[VI_Rules[L_i].Condition_Target_ID], 0.0, 1.0); END_IF;
                E_Rule_Condition_Type.COND_SMOKE: IF VI_Rules[L_i].Condition_Target_ID <= GVL_CONSTANTS.C_MAX_SMOKE_SENSORS THEN L_Current_Value := SEL(VI_Smoke_Sensors[VI_Rules[L_i].Condition_Target_ID], 0.0, 1.0); END_IF;
                E_Rule_Condition_Type.COND_METHANE: IF VI_Rules[L_i].Condition_Target_ID <= GVL_CONSTANTS.C_MAX_METHANE_SENSORS THEN L_Current_Value := VI_Methane_Sensors[VI_Rules[L_i].Condition_Target_ID]; END_IF;
                E_Rule_Condition_Type.COND_CO: IF VI_Rules[L_i].Condition_Target_ID <= GVL_CONSTANTS.C_MAX_CO_SENSORS THEN L_Current_Value := VI_CO_Sensors[VI_Rules[L_i].Condition_Target_ID]; END_IF;
                E_Rule_Condition_Type.COND_TIME_OF_DAY: L_Current_Value := TO_REAL(TOD_TO_UDINT(VI_Current_Time) / GVL_CONSTANTS.C_MS_IN_MINUTE);
                E_Rule_Condition_Type.COND_DAY_OF_WEEK: L_Current_Value := TO_REAL(VI_Day_Of_Week);
            END_CASE;
        ELSE
            IF VI_Rules[L_i].Condition_Type = E_Rule_Condition_Type.COND_TIME_OF_DAY THEN
                L_Current_Value := TO_REAL(TOD_TO_UDINT(VI_Current_Time) / GVL_CONSTANTS.C_MS_IN_MINUTE);
            ELSIF VI_Rules[L_i].Condition_Type = E_Rule_Condition_Type.COND_DAY_OF_WEEK THEN
                L_Current_Value := TO_REAL(VI_Day_Of_Week);
            END_IF;
        END_IF;

        CASE VI_Rules[L_i].Condition_Op OF
            E_Rule_Comparison.COMP_GT: L_Condition_Met := (L_Current_Value > VI_Rules[L_i].Condition_Value);
            E_Rule_Comparison.COMP_LT: L_Condition_Met := (L_Current_Value < VI_Rules[L_i].Condition_Value);
            E_Rule_Comparison.COMP_EQ: L_Condition_Met := (ABS(L_Current_Value - VI_Rules[L_i].Condition_Value) < 0.1);
            E_Rule_Comparison.COMP_GE: L_Condition_Met := (L_Current_Value >= VI_Rules[L_i].Condition_Value);
            E_Rule_Comparison.COMP_LE: L_Condition_Met := (L_Current_Value <= VI_Rules[L_i].Condition_Value);
            E_Rule_Comparison.COMP_IN_RANGE: L_Condition_Met := (L_Current_Value >= VI_Rules[L_i].Condition_Value) AND (L_Current_Value <= VI_Rules[L_i].Condition_Value_Max);
            E_Rule_Comparison.COMP_TRUE: L_Condition_Met := (L_Current_Value > 0.5);
            E_Rule_Comparison.COMP_FALSE: L_Condition_Met := (L_Current_Value < 0.5);
        END_CASE;

        L_Triggers[L_i](CLK := L_Condition_Met);

        IF L_Triggers[L_i].Q THEN
            L_Trigger_Count[L_i] := L_Trigger_Count[L_i] + 1;
            IF L_Trigger_Count[L_i] > 10 THEN
                VO_Actions[L_i].Active := FALSE;
                VO_Actions[L_i].Triggered := FALSE;
                CONTINUE;
            END_IF;
        END_IF;

        IF L_Condition_Met AND (L_Trigger_Count[L_i] <= 10) THEN
            VO_Actions[L_i].Active := TRUE;
            VO_Actions[L_i].Triggered := L_Triggers[L_i].Q;
            VO_Actions[L_i].Action_Type := VI_Rules[L_i].Action_Type;
            VO_Actions[L_i].Target_ID := VI_Rules[L_i].Action_Target_ID;
            VO_Actions[L_i].Value := VI_Rules[L_i].Action_Value;
        END_IF;
    END_IF;
END_FOR;

// >>> BULK_SYNC_ANCHOR: FB_Rule_Engine <<<

(* ---- FB_Safety_Workflow_Manager.st ---- *)
FUNCTION_BLOCK FB_Safety_Workflow_Manager
VAR_INPUT
    VI_System_Time_MS : UDINT;
    VI_Water_Selective_Recover : BOOL;
    VI_Gas_Selective_Recover : BOOL;
    VI_Water_Valve_Test_Open : BOOL;
    VI_Water_Valve_Test_Close : BOOL;
    VI_Water_Valve_Test_Confirm : BOOL;
    VI_Gas_Valve_Test_Open : BOOL;
    VI_Gas_Valve_Test_Close : BOOL;
    VI_Gas_Valve_Test_Confirm : BOOL;
END_VAR
VAR_OUTPUT
    VO_Water_Selective_Recover_Edge : BOOL;
    VO_Gas_Selective_Recover_Edge : BOOL;
    VO_Water_Valve_Test_Open_Edge : BOOL;
    VO_Water_Valve_Test_Close_Edge : BOOL;
    VO_Water_Valve_Test_Confirm_Edge : BOOL;
    VO_Gas_Valve_Test_Open_Edge : BOOL;
    VO_Gas_Valve_Test_Close_Edge : BOOL;
    VO_Gas_Valve_Test_Confirm_Edge : BOOL;
    VO_Water_Test_Active : BOOL;
    VO_Gas_Test_Active : BOOL;
    VO_Water_Test_Timeout_Close_Required : BOOL;
    VO_Gas_Test_Timeout_Close_Required : BOOL;
END_VAR
VAR
    L_CMD_Water_Selective_Recover_Prev : BOOL;
    L_CMD_Gas_Selective_Recover_Prev : BOOL;
    L_CMD_Water_Valve_Test_Open_Prev : BOOL;
    L_CMD_Water_Valve_Test_Close_Prev : BOOL;
    L_CMD_Water_Valve_Test_Confirm_Prev : BOOL;
    L_CMD_Gas_Valve_Test_Open_Prev : BOOL;
    L_CMD_Gas_Valve_Test_Close_Prev : BOOL;
    L_CMD_Gas_Valve_Test_Confirm_Prev : BOOL;
    L_Water_Test_Active : BOOL;
    L_Water_Test_Deadline : UDINT;
    L_Gas_Test_Active : BOOL;
    L_Gas_Test_Deadline : UDINT;
END_VAR

VO_Water_Test_Timeout_Close_Required := FALSE;
VO_Gas_Test_Timeout_Close_Required := FALSE;

VO_Water_Selective_Recover_Edge := VI_Water_Selective_Recover AND NOT L_CMD_Water_Selective_Recover_Prev;
VO_Gas_Selective_Recover_Edge := VI_Gas_Selective_Recover AND NOT L_CMD_Gas_Selective_Recover_Prev;
VO_Water_Valve_Test_Open_Edge := VI_Water_Valve_Test_Open AND NOT L_CMD_Water_Valve_Test_Open_Prev;
VO_Water_Valve_Test_Close_Edge := VI_Water_Valve_Test_Close AND NOT L_CMD_Water_Valve_Test_Close_Prev;
VO_Water_Valve_Test_Confirm_Edge := VI_Water_Valve_Test_Confirm AND NOT L_CMD_Water_Valve_Test_Confirm_Prev;
VO_Gas_Valve_Test_Open_Edge := VI_Gas_Valve_Test_Open AND NOT L_CMD_Gas_Valve_Test_Open_Prev;
VO_Gas_Valve_Test_Close_Edge := VI_Gas_Valve_Test_Close AND NOT L_CMD_Gas_Valve_Test_Close_Prev;
VO_Gas_Valve_Test_Confirm_Edge := VI_Gas_Valve_Test_Confirm AND NOT L_CMD_Gas_Valve_Test_Confirm_Prev;

L_CMD_Water_Selective_Recover_Prev := VI_Water_Selective_Recover;
L_CMD_Gas_Selective_Recover_Prev := VI_Gas_Selective_Recover;
L_CMD_Water_Valve_Test_Open_Prev := VI_Water_Valve_Test_Open;
L_CMD_Water_Valve_Test_Close_Prev := VI_Water_Valve_Test_Close;
L_CMD_Water_Valve_Test_Confirm_Prev := VI_Water_Valve_Test_Confirm;
L_CMD_Gas_Valve_Test_Open_Prev := VI_Gas_Valve_Test_Open;
L_CMD_Gas_Valve_Test_Close_Prev := VI_Gas_Valve_Test_Close;
L_CMD_Gas_Valve_Test_Confirm_Prev := VI_Gas_Valve_Test_Confirm;

IF VO_Water_Valve_Test_Open_Edge THEN
    L_Water_Test_Active := TRUE;
    L_Water_Test_Deadline := VI_System_Time_MS + 60000;
END_IF;

IF L_Water_Test_Active THEN
    IF VI_System_Time_MS >= L_Water_Test_Deadline THEN
        L_Water_Test_Active := FALSE;
        VO_Water_Test_Timeout_Close_Required := TRUE;
    END_IF;
END_IF;

IF VO_Gas_Valve_Test_Open_Edge THEN
    L_Gas_Test_Active := TRUE;
    L_Gas_Test_Deadline := VI_System_Time_MS + 60000;
END_IF;

IF L_Gas_Test_Active THEN
    IF VI_System_Time_MS >= L_Gas_Test_Deadline THEN
        L_Gas_Test_Active := FALSE;
        VO_Gas_Test_Timeout_Close_Required := TRUE;
    END_IF;
END_IF;

VO_Water_Test_Active := L_Water_Test_Active;
VO_Gas_Test_Active := L_Gas_Test_Active;
END_FUNCTION_BLOCK

(* ---- FB_Sensor_Analog_Processing.st ---- *)
FUNCTION_BLOCK FB_Sensor_Analog_Processing
VAR_INPUT
    VI_Raw_Value : WORD; // Raw value from module (e.g., 0-27648)
    VI_Sensor_Type : INT := 0; // 0: 4-20mA, 1: 0-10V, 2: PT100/1000 (direct temp * 10)
    VI_Min_Scale : REAL; // Minimum scale value (e.g., 0 bar)
    VI_Max_Scale : REAL; // Maximum scale value (e.g., 10 bar)
    VI_Offset : REAL; // Calibration offset
    VI_Multiplier : REAL := 1.0; // Calibration multiplier
    VI_Filter_Time_MS : UDINT := GVL_CONSTANTS.C_MS_IN_SECOND; // Filtering time
    VI_System_Time_MS : UDINT; // System time in ms
    VI_Fallback_Mode : INT := 0; // 0: Hold last good value, 1: Use default value
    VI_Default_Value : REAL := 0.0; // Default value for fallback mode 1
END_VAR
VAR_OUTPUT
    VO_Value : REAL; // Processed value
    VO_Error : BOOL; // Sensor error (open/short circuit)
    VO_Diag_Code : WORD; // Diagnostic code (0: OK, 1: Open circuit, 2: Short circuit, 3: Out of range)
END_VAR
VAR
    L_Scaled : REAL;
    L_Filtered : REAL;
    L_History : ARRAY[0..9] OF REAL; // Массив для скользящего среднего (10 значений)
    L_History_Idx : INT := 0;
    L_History_Sum : REAL := 0.0;
    L_History_Count : INT := 0;
    L_Last_Time : UDINT;
    L_DT : UDINT;
    L_First_Scan : BOOL := TRUE;
    L_i : INT;
END_VAR

// 1. Error checking and scaling based on sensor type
VO_Error := FALSE;
VO_Diag_Code := 0;

CASE VI_Sensor_Type OF
    0: // 4-20mA (NAMUR NE43: < 3.6mA or > 21mA)
        IF VI_Raw_Value < GVL_CONSTANTS.C_ANALOG_3_6MA_RAW THEN // < 3.6mA (Open circuit)
            VO_Error := TRUE;
            VO_Diag_Code := 1;
        ELSIF VI_Raw_Value > GVL_CONSTANTS.C_ANALOG_21MA_RAW THEN // > 21mA (Short circuit)
            VO_Error := TRUE;
            VO_Diag_Code := 2;
        ELSE
            // 4mA = 5529, 20mA = 27648
            L_Scaled := VI_Min_Scale + (TO_REAL(VI_Raw_Value - GVL_CONSTANTS.C_ANALOG_4MA_RAW) / TO_REAL(GVL_CONSTANTS.C_ANALOG_RAW_MAX - GVL_CONSTANTS.C_ANALOG_4MA_RAW)) * (VI_Max_Scale - VI_Min_Scale);
        END_IF;

    1: // 0-10V (0-27648)
        IF VI_Raw_Value > GVL_CONSTANTS.C_ANALOG_10V_MAX_RAW THEN // Out of range
            VO_Error := TRUE;
            VO_Diag_Code := 3;
        ELSE
            L_Scaled := VI_Min_Scale + (TO_REAL(VI_Raw_Value) / TO_REAL(GVL_CONSTANTS.C_ANALOG_RAW_MAX)) * (VI_Max_Scale - VI_Min_Scale);
        END_IF;

    2: // PT100/1000 (Direct temperature * 10, e.g., 255 = 25.5C)
        // Typically, 16-bit signed integer for temperature
        IF VI_Raw_Value = 16#7FFF OR VI_Raw_Value = 16#8000 THEN // Sensor error codes
            VO_Error := TRUE;
            VO_Diag_Code := 1;
        ELSE
            L_Scaled := TO_REAL(TO_INT(VI_Raw_Value)) / 10.0;
            IF L_Scaled < VI_Min_Scale OR L_Scaled > VI_Max_Scale THEN
                VO_Error := TRUE;
                VO_Diag_Code := 3;
            END_IF;
        END_IF;

    ELSE
        VO_Error := TRUE;
        VO_Diag_Code := 16#FFFF; // Unknown sensor type
END_CASE;

// 2. Fallback handling
IF VO_Error THEN
    IF VI_Fallback_Mode = 1 THEN
        VO_Value := VI_Default_Value;
    END_IF;
    // If VI_Fallback_Mode = 0, VO_Value retains its last good value (L_Filtered)
    RETURN;
END_IF;

// 3. Calibration
L_Scaled := (L_Scaled * VI_Multiplier) + VI_Offset;

// 4. Moving Average Filter (ТЗ 1.2)
IF L_First_Scan THEN
    L_Filtered := L_Scaled;
    L_First_Scan := FALSE;
    L_Last_Time := VI_System_Time_MS;

    // Инициализация массива истории
    FOR L_i := 0 TO 9 DO
        L_History[L_i] := L_Scaled;
    END_FOR;
    L_History_Sum := L_Scaled * 10.0;
    L_History_Count := 10;
    L_History_Idx := 0;
END_IF;

L_DT := (SEL(VI_System_Time_MS >= L_Last_Time, VI_System_Time_MS - L_Last_Time, (4294967295 - L_Last_Time) + VI_System_Time_MS + 1));
IF VI_Filter_Time_MS = 0 THEN
    L_Filtered := L_Scaled;
    L_Last_Time := VI_System_Time_MS;
ELSIF L_DT >= (VI_Filter_Time_MS / 10) THEN // Обновляем 10 раз за время фильтрации
    // Вычитаем старое значение
    L_History_Sum := L_History_Sum - L_History[L_History_Idx];

    // Добавляем новое значение
    L_History[L_History_Idx] := L_Scaled;
    L_History_Sum := L_History_Sum + L_Scaled;

    // Сдвигаем индекс
    L_History_Idx := (L_History_Idx + 1) MOD 10;

    // Вычисляем среднее
    L_Filtered := L_History_Sum / 10.0;

    L_Last_Time := VI_System_Time_MS;
END_IF;

VO_Value := L_Filtered;
END_FUNCTION_BLOCK

(* ---- FB_Smoke_Detector.st ---- *)
FUNCTION_BLOCK FB_Smoke_Detector
VAR_INPUT
    VI_Smoke_Signal : BOOL;
END_VAR
VAR_OUTPUT
    VO_Smoke_Detected : BOOL;
END_VAR

VO_Smoke_Detected := VI_Smoke_Signal;
END_FUNCTION_BLOCK

(* ---- FB_State_Replication.st ---- *)
FUNCTION_BLOCK FB_State_Replication
VAR_INPUT
    VI_Local_Role : E_PLC_ROLE; // Локальная роль ПЛК (Active/Standby)
    VI_Sync_Req : BOOL; // Запрос на принудительную синхронизацию
    VI_Local_State : ST_System_State_Snapshot; // Локальное состояние системы
    VI_Remote_State : ST_System_State_Snapshot; // Состояние системы партнера
    VI_System_Time_MS : UDINT; // Системное время (мс)
END_VAR
VAR_OUTPUT
    VO_State_Updated : BOOL; // Флаг: Состояние было обновлено
    VO_Synced_State : ST_System_State_Snapshot; // Синхронизированное состояние
END_VAR
VAR
    L_Sync_In_Progress : BOOL;
    L_Last_Sync_Time : UDINT;
    L_Periodic_Sync_Req : BOOL;
    L_Elapsed_Time : UDINT;
END_VAR

// Периодическая синхронизация (каждые 5 секунд)
L_Elapsed_Time := (SEL(VI_System_Time_MS >= L_Last_Sync_Time, VI_System_Time_MS - L_Last_Sync_Time, (4294967295 - L_Last_Sync_Time) + VI_System_Time_MS + 1));

IF L_Elapsed_Time > 5000 THEN
    L_Periodic_Sync_Req := TRUE;
    L_Last_Sync_Time := VI_System_Time_MS;
ELSE
    L_Periodic_Sync_Req := FALSE;
END_IF;

// State Replication Logic
// Синхронизация состояния между ПЛК (ТЗ 8.2)
IF (VI_Sync_Req OR L_Periodic_Sync_Req) AND NOT L_Sync_In_Progress THEN
    L_Sync_In_Progress := TRUE;

    // Разрешение конфликтов на основе версии состояния
    IF VI_Remote_State.Version > VI_Local_State.Version THEN
        VO_Synced_State := VI_Remote_State;
        VO_State_Updated := TRUE;
    ELSIF VI_Remote_State.Version = VI_Local_State.Version THEN
        // Если версии равны, приоритет у ведущего ПЛК
        IF VI_Local_Role = E_PLC_ROLE.ROLE_STANDBY THEN
            VO_Synced_State := VI_Remote_State;
            VO_State_Updated := TRUE;
        ELSE
            VO_Synced_State := VI_Local_State;
            VO_State_Updated := FALSE;
        END_IF;
    ELSE
        VO_Synced_State := VI_Local_State;
        VO_State_Updated := FALSE;
    END_IF;
ELSIF NOT (VI_Sync_Req OR L_Periodic_Sync_Req) THEN
    L_Sync_In_Progress := FALSE;
    VO_State_Updated := FALSE;
    VO_Synced_State := VI_Local_State;
END_IF;
END_FUNCTION_BLOCK

(* ---- FB_State_Snapshot_Manager.st ---- *)
FUNCTION_BLOCK FB_State_Snapshot_Manager
VAR_INPUT
    VI_System_Time_MS : UDINT;
    VI_Trigger_Event  : BOOL; // Сигнал на создание снимка
    VI_Event_Code     : WORD;
    VI_Current_State  : ST_State_Snapshot;
END_VAR
VAR_OUTPUT
    VO_Snapshot_Saved : BOOL;
END_VAR
VAR
    L_Snapshot_Buffer : ARRAY[1..GVL_CONSTANTS.C_MAX_STATE_SNAPSHOTS] OF ST_State_Snapshot;
    L_Write_Idx       : INT := 1;
END_VAR

IF VI_Trigger_Event THEN
    L_Snapshot_Buffer[L_Write_Idx] := VI_Current_State;
    L_Snapshot_Buffer[L_Write_Idx].timestamp_ms := VI_System_Time_MS;

    // NOTE:
    // ST_State_Snapshot no longer contains trigger_event_code in live project.
    // VI_Event_Code is reserved for future snapshot metadata extension.

    L_Write_Idx := (L_Write_Idx MOD GVL_CONSTANTS.C_MAX_STATE_SNAPSHOTS) + 1;
    VO_Snapshot_Saved := TRUE;
ELSE
    VO_Snapshot_Saved := FALSE;
END_IF;
END_FUNCTION_BLOCK

(* ---- FB_System_Coordinator.st ---- *)
FUNCTION_BLOCK FB_System_Coordinator

VAR_INPUT
    VI_Fire_Latched : BOOL;
    VI_Gas_Latched : BOOL;
    VI_Leak_Latched : BOOL;

    VI_IO_Degraded : BOOL;
    VI_Ownership_Violation : BOOL;

    VI_Behavior_Mode : E_Behavior_Mode;
END_VAR

VAR_OUTPUT
    VO_Block_Heating : BOOL;
    VO_Block_Ventilation : BOOL;
    VO_Block_Lighting : BOOL;
    VO_Block_Sockets : BOOL;

    VO_System_Degraded : BOOL;

    VO_Code : UDINT;
END_VAR

// reset
VO_Block_Heating := FALSE;
VO_Block_Ventilation := FALSE;
VO_Block_Lighting := FALSE;
VO_Block_Sockets := FALSE;
VO_System_Degraded := FALSE;
VO_Code := 0;

// FIRE has highest priority. Safety-stop ownership remains in PRG_Safety.
IF VI_Fire_Latched THEN
    VO_Block_Heating := TRUE;
    VO_Block_Ventilation := TRUE;
    VO_Block_Sockets := TRUE;
    VO_Code := 100;
    RETURN;
END_IF;

// GAS has higher priority than behavior mode.
IF VI_Gas_Latched THEN
    VO_Block_Heating := TRUE;
    VO_Block_Lighting := TRUE;
    VO_Block_Sockets := TRUE;
    VO_Code := 200;
    RETURN;
END_IF;

// LEAK blocks heating but does not suppress later degradation/mode overlays.
IF VI_Leak_Latched THEN
    VO_Block_Heating := TRUE;
    VO_Code := 300;
END_IF;

// IO degraded blocks heating and marks system degraded.
IF VI_IO_Degraded THEN
    VO_System_Degraded := TRUE;
    VO_Block_Heating := TRUE;
    IF VO_Code = 0 THEN
        VO_Code := 400;
    END_IF;
END_IF;

// Ownership violation marks system degraded. Test/result handler owns any safe-stop reaction.
IF VI_Ownership_Violation THEN
    VO_System_Degraded := TRUE;
    IF VO_Code = 0 THEN
        VO_Code := 500;
    END_IF;
END_IF;

// Behavior mode overlays. These are lower priority than safety/system faults.
CASE VI_Behavior_Mode OF
    BEHAVIOR_AWAY:
        VO_Block_Lighting := TRUE;
        VO_Block_Sockets := TRUE;
        IF VO_Code = 0 THEN
            VO_Code := 600;
        END_IF;

    BEHAVIOR_NIGHT:
        VO_Block_Lighting := TRUE;
        IF VO_Code = 0 THEN
            VO_Code := 700;
        END_IF;

    BEHAVIOR_MAINTENANCE:
        VO_Block_Heating := TRUE;
        VO_Block_Ventilation := TRUE;
        IF VO_Code = 0 THEN
            VO_Code := 800;
        END_IF;
END_CASE;

(* ---- FB_System_Evacuation.st ---- *)
// ==============================================================================
// System evacuation helper
//
// Internal helper for PRG_System.
// Owns evacuation guidance, target/hazard zone name projection,
// and evacuation lighting activation.
// ==============================================================================
FUNCTION_BLOCK FB_System_Evacuation
VAR
    L_i : INT;
END_VAR

FOR L_i := 1 TO 32 DO
    GVL_STATE.G_Evac_Guidance[L_i] := 0;

    IF GVL_STATE.G_Evac_Hazard_Zone[L_i] THEN
        GVL_STATE.G_Evac_Guidance[L_i] := -1;
    END_IF;

    IF GVL_CONFIG.G_Evac_Exit_Zones[L_i] AND NOT GVL_STATE.G_Evac_Hazard_Zone[L_i] THEN
        GVL_STATE.G_Evac_Guidance[L_i] := 1;
    END_IF;
END_FOR;

GVL_STATUS.G_Evac_Target_Zone_Name := '';
GVL_STATUS.G_Evac_Hazard_Zone_Name := '';

FOR L_i := 1 TO 32 DO
    IF (GVL_STATUS.G_Evac_Hazard_Zone_Name = '') AND GVL_STATE.G_Evac_Hazard_Zone[L_i] THEN
        GVL_STATUS.G_Evac_Hazard_Zone_Name := GVL_CONFIG.G_Evac_Zone_Names[L_i];
        IF GVL_STATUS.G_Evac_Hazard_Zone_Name = '' THEN
            GVL_STATUS.G_Evac_Hazard_Zone_Name := CONCAT('Zone ', INT_TO_STRING(L_i));
        END_IF;
    END_IF;

    IF (GVL_STATUS.G_Evac_Target_Zone_Name = '') AND (GVL_STATE.G_Evac_Guidance[L_i] = 1) THEN
        GVL_STATUS.G_Evac_Target_Zone_Name := GVL_CONFIG.G_Evac_Zone_Names[L_i];
        IF GVL_STATUS.G_Evac_Target_Zone_Name = '' THEN
            GVL_STATUS.G_Evac_Target_Zone_Name := CONCAT('Zone ', INT_TO_STRING(L_i));
        END_IF;
    END_IF;
END_FOR;

IF GVL_STATE.G_System_Mode = E_System_Operating_Mode.MODE_SAFE_STOP AND GVL_STATE.G_Safety_Smoke_Latched THEN
    GVL_STATE.G_Evacuation_Lighting_Active := TRUE;
ELSE
    GVL_STATE.G_Evacuation_Lighting_Active := FALSE;
END_IF;

// >>> BULK_SYNC_ANCHOR: FB_System_Evacuation <<<

(* ---- FB_System_Health.st ---- *)
FUNCTION_BLOCK FB_System_Health
VAR_INPUT
    VI_Smoke_Detected      : BOOL;
    VI_Gas_Detected        : BOOL;
    VI_CO_Warning_Level    : BOOL;
    VI_CO_Alarm_Level      : BOOL;
    VI_Leak_Detected       : BOOL;

    VI_Sensor_Fault        : BOOL := FALSE;
    VI_IO_Offline          : BOOL := FALSE;
    VI_Comm_Fault          : BOOL := FALSE;
    VI_Watchdog_Fault      : BOOL := FALSE;
    VI_Subsystem_Fault     : BOOL := FALSE;
END_VAR

VAR
    L_IO_Fault_Assert_Count        : UINT;
    L_IO_Fault_Clear_Count         : UINT;
    L_IO_Fault_Stable              : BOOL;

    L_Comm_Fault_Assert_Count      : UINT;
    L_Comm_Fault_Clear_Count       : UINT;
    L_Comm_Fault_Stable            : BOOL;

    L_Sensor_Fault_Assert_Count    : UINT;
    L_Sensor_Fault_Clear_Count     : UINT;
    L_Sensor_Fault_Stable          : BOOL;

    L_Subsystem_Assert_Count       : UINT;
    L_Subsystem_Clear_Count        : UINT;
    L_Subsystem_Fault_Stable       : BOOL;

    L_IO_Fault_Prev                : BOOL;
    L_Comm_Fault_Prev              : BOOL;
    L_Sensor_Fault_Prev            : BOOL;
    L_Subsystem_Fault_Prev         : BOOL;
    L_Watchdog_Fault_Prev          : BOOL;
END_VAR

VAR CONSTANT
    C_HEALTH_DEBOUNCE_CYCLES       : UINT := 3;
END_VAR

VAR_OUTPUT
    VO_System_Severity     : E_System_Severity;
    VO_Root_Cause          : E_System_Root_Cause;

    // compatibility outputs for existing orchestration
    VO_Sensor_Fault        : BOOL;
    VO_IO_Fault            : BOOL;
    VO_Comm_Fault          : BOOL;
    VO_Subsystem_Degraded  : BOOL;

    VO_First_Fault_Active  : BOOL;
    VO_First_Fault_Type    : INT;
    VO_First_Fault_Source  : INT;

    VO_IO_Fault_Count          : UDINT;
    VO_Comm_Fault_Count        : UDINT;
    VO_Sensor_Fault_Count      : UDINT;
    VO_Subsystem_Fault_Count   : UDINT;
    VO_Watchdog_Fault_Count    : UDINT;
END_VAR

// Debounce non-critical diagnostics: require 3 stable cycles to assert/clear
IF VI_IO_Offline THEN
    L_IO_Fault_Clear_Count := 0;
    IF L_IO_Fault_Assert_Count < C_HEALTH_DEBOUNCE_CYCLES THEN
        L_IO_Fault_Assert_Count := L_IO_Fault_Assert_Count + 1;
    END_IF;
    IF L_IO_Fault_Assert_Count >= C_HEALTH_DEBOUNCE_CYCLES THEN
        L_IO_Fault_Stable := TRUE;
    END_IF;
ELSE
    L_IO_Fault_Assert_Count := 0;
    IF L_IO_Fault_Clear_Count < C_HEALTH_DEBOUNCE_CYCLES THEN
        L_IO_Fault_Clear_Count := L_IO_Fault_Clear_Count + 1;
    END_IF;
    IF L_IO_Fault_Clear_Count >= C_HEALTH_DEBOUNCE_CYCLES THEN
        L_IO_Fault_Stable := FALSE;
    END_IF;
END_IF;

IF VI_Comm_Fault THEN
    L_Comm_Fault_Clear_Count := 0;
    IF L_Comm_Fault_Assert_Count < C_HEALTH_DEBOUNCE_CYCLES THEN
        L_Comm_Fault_Assert_Count := L_Comm_Fault_Assert_Count + 1;
    END_IF;
    IF L_Comm_Fault_Assert_Count >= C_HEALTH_DEBOUNCE_CYCLES THEN
        L_Comm_Fault_Stable := TRUE;
    END_IF;
ELSE
    L_Comm_Fault_Assert_Count := 0;
    IF L_Comm_Fault_Clear_Count < C_HEALTH_DEBOUNCE_CYCLES THEN
        L_Comm_Fault_Clear_Count := L_Comm_Fault_Clear_Count + 1;
    END_IF;
    IF L_Comm_Fault_Clear_Count >= C_HEALTH_DEBOUNCE_CYCLES THEN
        L_Comm_Fault_Stable := FALSE;
    END_IF;
END_IF;

IF VI_Sensor_Fault THEN
    L_Sensor_Fault_Clear_Count := 0;
    IF L_Sensor_Fault_Assert_Count < C_HEALTH_DEBOUNCE_CYCLES THEN
        L_Sensor_Fault_Assert_Count := L_Sensor_Fault_Assert_Count + 1;
    END_IF;
    IF L_Sensor_Fault_Assert_Count >= C_HEALTH_DEBOUNCE_CYCLES THEN
        L_Sensor_Fault_Stable := TRUE;
    END_IF;
ELSE
    L_Sensor_Fault_Assert_Count := 0;
    IF L_Sensor_Fault_Clear_Count < C_HEALTH_DEBOUNCE_CYCLES THEN
        L_Sensor_Fault_Clear_Count := L_Sensor_Fault_Clear_Count + 1;
    END_IF;
    IF L_Sensor_Fault_Clear_Count >= C_HEALTH_DEBOUNCE_CYCLES THEN
        L_Sensor_Fault_Stable := FALSE;
    END_IF;
END_IF;

IF VI_Subsystem_Fault THEN
    L_Subsystem_Clear_Count := 0;
    IF L_Subsystem_Assert_Count < C_HEALTH_DEBOUNCE_CYCLES THEN
        L_Subsystem_Assert_Count := L_Subsystem_Assert_Count + 1;
    END_IF;
    IF L_Subsystem_Assert_Count >= C_HEALTH_DEBOUNCE_CYCLES THEN
        L_Subsystem_Fault_Stable := TRUE;
    END_IF;
ELSE
    L_Subsystem_Assert_Count := 0;
    IF L_Subsystem_Clear_Count < C_HEALTH_DEBOUNCE_CYCLES THEN
        L_Subsystem_Clear_Count := L_Subsystem_Clear_Count + 1;
    END_IF;
    IF L_Subsystem_Clear_Count >= C_HEALTH_DEBOUNCE_CYCLES THEN
        L_Subsystem_Fault_Stable := FALSE;
    END_IF;
END_IF;

// Count confirmed fault events on rising edge of stable/critical conditions
IF L_IO_Fault_Stable AND NOT L_IO_Fault_Prev THEN
    VO_IO_Fault_Count := VO_IO_Fault_Count + 1;
END_IF;
L_IO_Fault_Prev := L_IO_Fault_Stable;

IF L_Comm_Fault_Stable AND NOT L_Comm_Fault_Prev THEN
    VO_Comm_Fault_Count := VO_Comm_Fault_Count + 1;
END_IF;
L_Comm_Fault_Prev := L_Comm_Fault_Stable;

IF L_Sensor_Fault_Stable AND NOT L_Sensor_Fault_Prev THEN
    VO_Sensor_Fault_Count := VO_Sensor_Fault_Count + 1;
END_IF;
L_Sensor_Fault_Prev := L_Sensor_Fault_Stable;

IF L_Subsystem_Fault_Stable AND NOT L_Subsystem_Fault_Prev THEN
    VO_Subsystem_Fault_Count := VO_Subsystem_Fault_Count + 1;
END_IF;
L_Subsystem_Fault_Prev := L_Subsystem_Fault_Stable;

IF VI_Watchdog_Fault AND NOT L_Watchdog_Fault_Prev THEN
    VO_Watchdog_Fault_Count := VO_Watchdog_Fault_Count + 1;
END_IF;
L_Watchdog_Fault_Prev := VI_Watchdog_Fault;

VO_Sensor_Fault := L_Sensor_Fault_Stable;
VO_IO_Fault := L_IO_Fault_Stable;
VO_Comm_Fault := L_Comm_Fault_Stable;
VO_Subsystem_Degraded := L_Subsystem_Fault_Stable;

VO_System_Severity := E_System_Severity.SEV_NORMAL;
VO_Root_Cause := E_System_Root_Cause.ROOT_NONE;
VO_First_Fault_Active := FALSE;
VO_First_Fault_Type := 0;
VO_First_Fault_Source := 0;

// Priority: FIRE > GAS > CO > WATER > diagnostics
IF VI_Smoke_Detected THEN
    VO_System_Severity := E_System_Severity.SEV_CRITICAL;
    VO_Root_Cause := E_System_Root_Cause.ROOT_FIRE;
    VO_First_Fault_Active := TRUE;
    VO_First_Fault_Type := 5;

ELSIF VI_Gas_Detected THEN
    VO_System_Severity := E_System_Severity.SEV_CRITICAL;
    VO_Root_Cause := E_System_Root_Cause.ROOT_GAS_LEAK;
    VO_First_Fault_Active := TRUE;
    VO_First_Fault_Type := 6;

ELSIF VI_CO_Alarm_Level THEN
    VO_System_Severity := E_System_Severity.SEV_CRITICAL;
    VO_Root_Cause := E_System_Root_Cause.ROOT_CO_CRITICAL;
    VO_First_Fault_Active := TRUE;
    VO_First_Fault_Type := 7;

ELSIF VI_CO_Warning_Level THEN
    VO_System_Severity := E_System_Severity.SEV_WARNING;
    VO_Root_Cause := E_System_Root_Cause.ROOT_CO_WARNING;
    VO_First_Fault_Active := TRUE;
    VO_First_Fault_Type := 7;

ELSIF VI_Leak_Detected THEN
    VO_System_Severity := E_System_Severity.SEV_WARNING;
    VO_Root_Cause := E_System_Root_Cause.ROOT_WATER_LEAK;
    VO_First_Fault_Active := TRUE;
    VO_First_Fault_Type := 8;

ELSIF VI_Watchdog_Fault THEN
    VO_System_Severity := E_System_Severity.SEV_CRITICAL;
    VO_Root_Cause := E_System_Root_Cause.ROOT_WATCHDOG_FAULT;
    VO_First_Fault_Active := TRUE;
    VO_First_Fault_Type := 9;

ELSIF L_IO_Fault_Stable THEN
    VO_System_Severity := E_System_Severity.SEV_DEGRADED;
    VO_Root_Cause := E_System_Root_Cause.ROOT_IO_OFFLINE;
    VO_First_Fault_Active := TRUE;
    VO_First_Fault_Type := 1;

ELSIF L_Comm_Fault_Stable THEN
    VO_System_Severity := E_System_Severity.SEV_DEGRADED;
    VO_Root_Cause := E_System_Root_Cause.ROOT_COMM_FAULT;
    VO_First_Fault_Active := TRUE;
    VO_First_Fault_Type := 3;

ELSIF L_Sensor_Fault_Stable THEN
    VO_System_Severity := E_System_Severity.SEV_DEGRADED;
    VO_Root_Cause := E_System_Root_Cause.ROOT_SENSOR_FAULT;
    VO_First_Fault_Active := TRUE;
    VO_First_Fault_Type := 2;

ELSIF L_Subsystem_Fault_Stable THEN
    VO_System_Severity := E_System_Severity.SEV_DEGRADED;
    VO_Root_Cause := E_System_Root_Cause.ROOT_SUBSYSTEM_FAULT;
    VO_First_Fault_Active := TRUE;
    VO_First_Fault_Type := 4;
END_IF;
// >>> BULK_SYNC_ANCHOR: FB_System_Health <<<
END_FUNCTION_BLOCK

(* ---- FB_System_Intent_Publisher.st ---- *)
// ==============================================================================
// System intent publisher helper
//
// Internal helper for PRG_System.
// Owns publication of system-mode gates into GVL_INTENT_SYSTEM.
// ==============================================================================
FUNCTION_BLOCK FB_System_Intent_Publisher
VAR_INPUT
    VI_System_Time_MS : UDINT;
    VI_Gateway_Writes_Allowed : BOOL;
END_VAR

GVL_INTENT_SYSTEM.I_Source_Valid := TRUE;
GVL_INTENT_SYSTEM.I_Last_Update_MS := VI_System_Time_MS;
GVL_INTENT_SYSTEM.I_Mode_Safe_Stop_Active := (GVL_STATE.G_System_Mode = E_System_Operating_Mode.MODE_SAFE_STOP);
GVL_INTENT_SYSTEM.I_Mode_Degraded_Active := (GVL_STATE.G_System_Mode = E_System_Operating_Mode.MODE_DEGRADED);
GVL_INTENT_SYSTEM.I_Mode_Freeze_Protection_Active := (GVL_STATE.G_System_Mode = E_System_Operating_Mode.MODE_FREEZE_PROTECTION);
GVL_INTENT_SYSTEM.I_Operator_Scenario_Block := (GVL_STATE.G_System_Mode = E_System_Operating_Mode.MODE_SAFE_STOP);
GVL_INTENT_SYSTEM.I_Lighting_Overrides_Block := (GVL_STATE.G_System_Mode = E_System_Operating_Mode.MODE_SAFE_STOP);
GVL_INTENT_SYSTEM.I_Blinds_Overrides_Block := (GVL_STATE.G_System_Mode = E_System_Operating_Mode.MODE_SAFE_STOP);
GVL_INTENT_SYSTEM.I_Socket_Overrides_Block := (GVL_STATE.G_System_Mode = E_System_Operating_Mode.MODE_SAFE_STOP);
GVL_INTENT_SYSTEM.I_Gateway_Writes_Allowed := VI_Gateway_Writes_Allowed;
GVL_INTENT_SYSTEM.I_Scenario_Request_Allowed := (GVL_STATE.G_System_Mode <> E_System_Operating_Mode.MODE_SAFE_STOP);

// >>> BULK_SYNC_ANCHOR: FB_System_Intent_Publisher <<<
END_FUNCTION_BLOCK

(* ---- FB_System_Recovery.st ---- *)
// ==============================================================================
// System recovery helper
//
// Internal helper for PRG_System.
// Owns one-shot recovery of persistent safety/system state after boot.
// ==============================================================================
FUNCTION_BLOCK FB_System_Recovery
VAR_IN_OUT
    VIO_Recovery_Done : BOOL;
END_VAR

IF NOT VIO_Recovery_Done THEN
    IF GVL_PERSISTENT.P_Valid THEN
        GVL_STATE.G_Safety_Gas_Latched := GVL_PERSISTENT.P_Safety_Gas_Latched;
        GVL_STATE.G_Safety_Smoke_Latched := GVL_PERSISTENT.P_Safety_Smoke_Latched;
        GVL_STATE.G_Safety_Leak_Latched := GVL_PERSISTENT.P_Safety_Leak_Latched;
        GVL_STATE.G_System_Mode := GVL_PERSISTENT.P_System_Mode;
    END_IF;

    VIO_Recovery_Done := TRUE;
END_IF;

// >>> BULK_SYNC_ANCHOR: FB_System_Recovery <<<
END_FUNCTION_BLOCK

(* ---- FB_System_Redundancy_Orchestrator.st ---- *)
// ==============================================================================
// System redundancy orchestrator helper
//
// Internal helper for PRG_System.
// Owns PLC role calculation, heartbeat output projection, and synced-state apply.
// ==============================================================================
FUNCTION_BLOCK FB_System_Redundancy_Orchestrator
VAR_IN_OUT
    VIO_Local_State : ST_System_State_Snapshot;
    VIO_Remote_State : ST_System_State_Snapshot;
END_VAR

VAR
    fbRedundancy : FB_Redundancy_Manager;
END_VAR

// Build local state snapshot for replication.
VIO_Local_State.System_Time_MS := GVL_STATUS.G_System_Time_MS;
VIO_Local_State.Current_Scenario := GVL_STATUS.G_Current_Scenario;
VIO_Local_State.Security_Armed := GVL_ALARM.G_Security_Armed;
VIO_Local_State.Active_Alarms := GVL_ALARM.G_Active_Alarm_Count;
VIO_Local_State.Zone_Valves := GVL_STATE.G_Zone_Valves;
VIO_Local_State.Manifold_Pumps := GVL_STATE.G_Manifold_Pumps;
VIO_Local_State.Lighting_States := GVL_STATE.G_Lighting_Levels;
VIO_Local_State.Blinds_Positions := GVL_STATE.G_Blinds_Positions;
VIO_Local_State.Socket_States := GVL_STATE.G_Socket_States;
VIO_Local_State.Gas_Valve_Closed := GVL_COMMAND.G_Gas_Valve_Close;
VIO_Local_State.Water_Valves_Closed := GVL_COMMAND.G_Close_Valve_36;
VIO_Local_State.Version := VIO_Local_State.Version + 1;

fbRedundancy(
    VI_System_Time_MS := GVL_STATUS.G_System_Time_MS,
    VI_Local_PLC_ID := GVL_STATUS.G_PLC_ID,
    VI_Remote_Pulse := GVL_IO.DI_Partner_Pulse,
    VI_Remote_Is_Active := GVL_IO.DI_Partner_Active,
    VI_Gateway_Ping_OK := GVL_GATEWAY.G_Gateway_Ping_OK,
    VI_Local_State := VIO_Local_State,
    VI_Remote_State := VIO_Remote_State
);

GVL_STATUS.G_Is_Active_PLC := (fbRedundancy.VO_Local_Role = E_PLC_ROLE.ROLE_ACTIVE);
GVL_IO.DO_Heartbeat_Pulse := fbRedundancy.VO_Local_Pulse;
GVL_IO.DO_Active_Status := GVL_STATUS.G_Is_Active_PLC;

IF fbRedundancy.VO_State_Updated THEN
    GVL_STATUS.G_Current_Scenario := fbRedundancy.VO_Synced_State.Current_Scenario;
    GVL_ALARM.G_Security_Armed := fbRedundancy.VO_Synced_State.Security_Armed;
    GVL_STATE.G_Zone_Valves := fbRedundancy.VO_Synced_State.Zone_Valves;
    GVL_STATE.G_Manifold_Pumps := fbRedundancy.VO_Synced_State.Manifold_Pumps;
    GVL_STATE.G_Lighting_Levels := fbRedundancy.VO_Synced_State.Lighting_States;
    GVL_STATE.G_Blinds_Positions := fbRedundancy.VO_Synced_State.Blinds_Positions;
    GVL_STATE.G_Socket_States := fbRedundancy.VO_Synced_State.Socket_States;
    GVL_COMMAND.G_Gas_Valve_Close := fbRedundancy.VO_Synced_State.Gas_Valve_Closed;
    GVL_COMMAND.G_Close_Valve_36 := fbRedundancy.VO_Synced_State.Water_Valves_Closed;
    VIO_Local_State.Version := fbRedundancy.VO_Synced_State.Version;
END_IF;

// >>> BULK_SYNC_ANCHOR: FB_System_Redundancy_Orchestrator <<<
